	(*Part 37 Present*)
		Part_Present37FB(
			Sensor_Input:= N08.I.4,
			On_Trigger1:= Enable_Motion AND In_Auto AND NOT Unload_Complete,
			On_Trigger2:= TRUE,
			Off_Trigger1:= Dry_Cycle OR (Cycle_Complete  AND NOT Enable_Motion),
			Off_Trigger2:= TRUE,
			Disable_Faults:= FALSE,
			Fault_Delay:= T#1.5s,
			Status=> Part_Present37,
			Faulted=>  PPFaults1.8);

	(*Part 38 Present*)
		Part_Present38FB(
			Sensor_Input:= N08.I.5,
			On_Trigger1:= Enable_Motion AND In_Auto AND NOT Unload_Complete,
			On_Trigger2:= TRUE,
			Off_Trigger1:= Dry_Cycle OR (Cycle_Complete  AND NOT Enable_Motion),
			Off_Trigger2:= TRUE,
			Disable_Faults:= FALSE,
			Fault_Delay:= T#1.5s,
			Status=> Part_Present38,
			Faulted=>  PPFaults1.9);

	(*Part 39 Present*)
		Part_Present39FB(
			Sensor_Input:= N08.I.6,
			On_Trigger1:= Enable_Motion AND In_Auto AND NOT Unload_Complete,
			On_Trigger2:= TRUE,
			Off_Trigger1:= Dry_Cycle OR (Cycle_Complete  AND NOT Enable_Motion),
			Off_Trigger2:= TRUE,
			Disable_Faults:= FALSE,
			Fault_Delay:= T#1.5s,
			Status=> Part_Present39,
			Faulted=>  PPFaults1.10);

	(*Part 40 Present*)
		Part_Present40FB(
			Sensor_Input:= N08.I.7,
			On_Trigger1:= Enable_Motion AND In_Auto AND NOT Unload_Complete,
			On_Trigger2:= TRUE,
			Off_Trigger1:= Dry_Cycle OR (Cycle_Complete  AND NOT Enable_Motion),
			Off_Trigger2:= TRUE,
			Disable_Faults:= FALSE,
			Fault_Delay:= T#1.5s,
			Status=> Part_Present40,
			Faulted=>  PPFaults1.11);



(*end*)
END_ACTION

ACTION Robot_Registration:


(*#################################### Register Robots to Tool ##################################*)
(*+++++++++++THIS AREA IS CUSTOM PER INSTALLATION AND WILL HAVE TO BE MODIFIED PER +++++++++++++*)
(*+++++++++++THIS AREA IS CUSTOM PER INSTALLATION AND WILL HAVE TO BE MODIFIED PER +++++++++++++*)
(*NOTE: See Example code in Fix 15 / 16*)
(*NOTE: See Example code in Fix 15 / 16*)

	(*Data From Load Robot(s)*)
	Load_Robots_Clear1:= TRUE;
	Load_Robots_Clear2:= TRUE;
	Load_Robots_Clear:=Load_Robots_Clear1 AND Load_Robots_Clear2;
	Load_Robots_WorkingOK1:= FALSE;
	Load_Robots_WorkingOK2:= FALSE;
	IF FALSE
		THEN
		Load_Robots_UnclampEarly1:= TRUE;
	END_IF;
	IF FALSE
		THEN
		Load_Robots_UnclampEarly2:= TRUE;
	END_IF;
	Load_Robots_Complete1:= FALSE;
	Load_Robots_Complete2:= FALSE;
	Load_Robots_PartInEOAT1:= FALSE;
	Load_Robots_PartInEOAT2:= FALSE;


	(*Data From Turntable*)
	TurntableA_Clear:= TRUE;
	TurntableB_Clear:= TRUE;
	Turntable_Clear:= TurntableA_Clear AND TurntableB_Clear;
	TurntableA_At_Robot:= FALSE;
	TurntableB_At_Robot:= FALSE;
	Turntable_WorkingOK:= FALSE;
	TurntableA_Complete:= FALSE;
	TurntableB_Complete:= FALSE;


	(*Data From Seal Robot(s)*)
	Seal_Robots_Clear:= TRUE;
	Seal_Robots_WorkingOK:= FALSE;
	IF FALSE
		THEN
		Seal_Robots_UnclampEarly:= TRUE;
	END_IF;
	Seal_Robots_Complete:= FALSE;


	(*Data From Stud Robot(s)*)
	Stud_Robots_Clear:= TRUE;
	Stud_Robots_WorkingOK:= FALSE;
	IF FALSE
		THEN
		Stud_Robots_UnclampEarly:= TRUE;
	END_IF;
	Stud_Robots_Complete:= FALSE;


	(*Data From Weld Robot(s)*)
	Weld_Robots_Clear:= TRUE;
	Weld_Robots_WorkingOK:= FALSE;
	IF FALSE
		THEN
		Weld_Robots_UnclampEarly:= TRUE;
	END_IF;
	Weld_Robots_Complete:= FALSE;

	(*Change Robots for Current Fixture functionality*) (*If no MIG robots Set to True.  Example code is in Fix15/16*) 
	Mig_Robots_Ready:=	TRUE; 

	(*Data From Unload Robot(s)*)
	Unload_Robots_Clear1:= TRUE;
	Unload_Robots_Clear2:= TRUE;
	Unload_Robots_Clear:= Unload_Robots_Clear1 AND Unload_Robots_Clear2;
	Unload_Robots_WorkingOK1:= FALSE;
	Unload_Robots_WorkingOK2:= FALSE;
	Unload_Robots_Complete1:= FALSE;
	Unload_Robots_Complete2:= FALSE;
	Unload_Robots_EOATEmpty1:=FALSE;
	Unload_Robots_EOATEmpty2:= FALSE;



	(*Amalgumate All Robots Clear of Tool*)
	All_Robots_Clear:= Load_Robots_Clear AND Seal_Robots_Clear AND Stud_Robots_Clear AND Turntable_Clear AND Weld_Robots_Clear AND Unload_Robots_Clear;

	(*Data To All Robots*)
	(*Task ID*)
	R1_Data.Task_ID[1]:=Task_ID;

	(*Fix ID*)
	R1_Data.Fix_ID[1]:=Fix_ID;

	(*Model ID*)
	R1_Data.Model_ID[1]:=Model_ID;

	(*Proceed from Pounce*)
	R1_Data.Proceed_From_Pounce[1]:= Robots_Clear_ToProceed;

	(*Complete Acks*)
	R1_Data.Complete_Ack[1]:=(Weld_Complete_Ack AND Weld_Robots_WorkingOK);

	(*Repo Acks*)
	R1_Data.PeripheralReq_Ack[1]:= Repo_Ack;

(*%%%%%%%%%%%%%% Call Robots to Tool and Give Them, Task ID, Fixture ID and Model ID %%%%%%%%%%%%%%%%%*)
	(* Perform Call To Tool*)
	Tool_Call_ForLoadRobots1:= Enable_Motion AND (NOT Cell_In_Services OR NOT Load_Robots_Clear1)
						AND Start_Load_Robots1 AND NOT Start_Load_Robots2 AND NOT Start_Weld_Robots AND NOT Start_Seal_Robots AND NOT Start_Stud_Robots
						AND NOT Start_Unload_Robots1 AND NOT Start_Unload_Robots2 AND NOT Start_TurntableA AND NOT Start_TurntableB;
	Tool_Call_ForLoadRobots2:= Enable_Motion AND (NOT Cell_In_Services OR NOT Load_Robots_Clear2)
						AND NOT Start_Load_Robots1 AND Start_Load_Robots2 AND NOT Start_Weld_Robots AND NOT Start_Seal_Robots AND NOT Start_Stud_Robots
						AND NOT Start_Unload_Robots1 AND NOT Start_Unload_Robots2 AND NOT Start_TurntableA AND NOT Start_TurntableB;
	Tool_Call_ForSealRobots:=Enable_Motion AND (NOT Cell_In_Services OR NOT Seal_Robots_Clear)
						AND NOT Start_Load_Robots1 AND NOT Start_Load_Robots2 AND NOT Start_Weld_Robots AND Start_Seal_Robots AND NOT Start_Stud_Robots
						AND NOT Start_Unload_Robots1 AND NOT Start_Unload_Robots2 AND NOT Start_TurntableA AND NOT Start_TurntableB;
	Tool_Call_ForStudRobots:=Enable_Motion AND (NOT Cell_In_Services OR NOT Stud_Robots_Clear)
						AND NOT Start_Load_Robots1 AND NOT Start_Load_Robots2 AND NOT Start_Weld_Robots AND NOT Start_Seal_Robots AND Start_Stud_Robots
						AND NOT Start_Unload_Robots1 AND NOT Start_Unload_Robots2 AND NOT Start_TurntableA AND NOT Start_TurntableB;
	Tool_Call_ForSweepA:= Enable_Motion AND (NOT Cell_In_Services OR NOT TurntableA_Clear)
						AND NOT Start_Load_Robots1 AND NOT Start_Load_Robots2 AND NOT Start_Weld_Robots AND NOT Start_Seal_Robots AND NOT Start_Stud_Robots
						AND NOT Start_Unload_Robots1 AND NOT Start_Unload_Robots2 AND Start_TurntableA AND NOT Start_TurntableB;
	Tool_Call_ForSweepB:= Enable_Motion AND (NOT Cell_In_Services OR NOT TurntableB_Clear)
						AND NOT Start_Load_Robots1 AND NOT Start_Load_Robots2 AND NOT Start_Weld_Robots AND NOT Start_Seal_Robots AND NOT Start_Stud_Robots
						AND NOT Start_Unload_Robots1 AND NOT Start_Unload_Robots2 AND NOT Start_TurntableA AND Start_TurntableB;
	Tool_Call_ForWeldRobots:= Enable_Motion AND (NOT Cell_In_Services OR NOT Weld_Robots_Clear)
						AND NOT Start_Load_Robots1 AND NOT Start_Load_Robots2 AND Start_Weld_Robots AND NOT Start_Seal_Robots AND NOT Start_Stud_Robots
						AND NOT Start_Unload_Robots1 AND NOT Start_Unload_Robots2 AND NOT Start_TurntableA AND NOT Start_TurntableB;
	Tool_Call_ForUnloadRobots1:= Enable_Motion AND (NOT Cell_In_Services OR NOT Unload_Robots_Clear1)
						AND NOT Start_Load_Robots1 AND NOT Start_Load_Robots2 AND NOT Start_Weld_Robots AND NOT Start_Seal_Robots AND NOT Start_Stud_Robots
						AND Start_Unload_Robots1 AND NOT Start_Unload_Robots2 AND NOT Start_TurntableA AND NOT Start_TurntableB;
	Tool_Call_ForUnloadRobots2:= Enable_Motion AND (NOT Cell_In_Services OR NOT Unload_Robots_Clear2)
						AND NOT Start_Load_Robots1 AND NOT Start_Load_Robots2 AND NOT Start_Weld_Robots AND NOT Start_Seal_Robots AND NOT Start_Stud_Robots
						AND NOT Start_Unload_Robots1 AND Start_Unload_Robots2 AND NOT Start_TurntableA AND NOT Start_TurntableB;



	(*Allow Robots to Proceed Into Tool*)
	(*!!!!!This is the final OK to allow Robots Into the Tool Area, So it Better Be Ready!!!!!!!*)
	IF Enable_Motion
		THEN
			IF Load_Robots_Proceed1 AND Load_Robots_WorkingOK1 AND Load_Robots_Clear2 AND Seal_Robots_Clear AND Stud_Robots_Clear AND Turntable_Clear AND Weld_Robots_Clear AND Unload_Robots_Clear
				THEN Robots_Clear_ToProceed:=TRUE;
			ELSIF Load_Robots_Proceed2 AND Load_Robots_WorkingOK2 AND Load_Robots_Clear1 AND Seal_Robots_Clear AND Stud_Robots_Clear AND Turntable_Clear AND Weld_Robots_Clear AND Unload_Robots_Clear
				THEN Robots_Clear_ToProceed:=TRUE;
			ELSIF Seal_Robots_Proceed AND Seal_Robots_WorkingOK AND Load_Robots_Clear AND Stud_Robots_Clear AND Turntable_Clear AND Weld_Robots_Clear AND Unload_Robots_Clear
				THEN Robots_Clear_ToProceed:=TRUE;
			ELSIF Stud_Robots_Proceed AND Stud_Robots_WorkingOK AND Load_Robots_Clear AND Seal_Robots_Clear AND Turntable_Clear AND Weld_Robots_Clear AND Unload_Robots_Clear
				THEN Robots_Clear_ToProceed:=TRUE;
			ELSIF Weld_Robots_Proceed AND Weld_Robots_WorkingOK AND Load_Robots_Clear AND Seal_Robots_Clear AND Stud_Robots_Clear AND Turntable_Clear AND Unload_Robots_Clear
				THEN Robots_Clear_ToProceed:=TRUE;
			ELSIF Unload_Robots_Proceed1 AND Unload_Robots_WorkingOK1 AND Load_Robots_Clear AND Seal_Robots_Clear AND Stud_Robots_Clear AND Turntable_Clear AND Weld_Robots_Clear AND Unload_Robots_Clear2
				THEN Robots_Clear_ToProceed:=TRUE;
			ELSIF Unload_Robots_Proceed2 AND Unload_Robots_WorkingOK2 AND Load_Robots_Clear AND Seal_Robots_Clear AND Stud_Robots_Clear AND Turntable_Clear AND Weld_Robots_Clear AND Unload_Robots_Clear1
				THEN Robots_Clear_ToProceed:=TRUE;
			ELSE Robots_Clear_ToProceed:= FALSE;
			END_IF;
		ELSE Robots_Clear_ToProceed:= FALSE;
	END_IF;

(*+++++++++++++++++++++++++++++++++++++++++++++++ Task Complete Acks ++++++++++++++++++++++++++*)
	(*1st Load Complete Ack*)
	Load_Complete1_Ack:= Load_Robots_Complete1 AND Load_Complete1;

	(*2nd Load Complete Ack*)
	Load_Complete2_Ack:= Load_Robots_Complete2 AND Load_Complete2;

	(*Seal Complete Ack*)
	Seal_Complete_Ack:= Seal_Robots_Complete AND Sealing_Complete;

	(*Stud Complete Ack*)
	Stud_Complete_Ack:= Stud_Robots_Complete AND Stud_Complete;

	(*Sweep Complete ACK*)
	TurnA_Complete_Ack := TurntableA_Complete AND TurntableA_At_Robot;
	TurnB_Complete_Ack := TurntableB_Complete AND TurntableB_At_Robot;

	(*Weld Complete Ack*)
	Weld_Complete_Ack:= Weld_Robots_Complete AND Welding_Complete;

	(*Unload Complete Ack*)
	Unload_Complete1_Ack:= Unload_Robots_Complete1 AND Unload_Complete;

	(*Unload Complete Ack*)
	Unload_Complete2_Ack:= Unload_Robots_Complete2 AND Unload_Complete;







(*end*)
END_ACTION

ACTION Status_and_Faults:



(*^^^^^^^^^^^^^^^^^^^^^^^^^^^^^^^^^^^^^^ General Visualization ^^^^^^^^^^^^^^^^^^^^^^^^^^^^^^^^^^^^*)
	(*For Ready to Load Indicators*)
		(*Flash when tool should be loaded but load is not complete*)
		IF In_Auto AND Tool_At_Home AND NOT Welding_Complete AND All_Robots_Clear AND NOT All_Sensors_On.2
			THEN
				Ready_To_Load:= Pulse_500mS;
				(*Go solid when tool has been loaded properly*)
				(*Go solid when tool is ready to be unloaded*)
		ELSIF In_Auto AND All_Robots_Clear  AND ((Tool_At_Home AND NOT Welding_Complete AND All_Sensors_On.2 AND NOT Enable_Motion)
			OR (Tool_At_Unload.0 AND Welding_Complete AND (Sealing_Complete OR Sealer_Bypass) AND (Stud_Complete OR Stud_Bypass) AND TurntableA_At_Robot AND NOT All_Sensors_Off))
			THEN
				Ready_To_Load:= TRUE;
		ELSE
				Ready_To_Load:= FALSE;
		END_IF;
	(*For Red Stack Light Indicators*)
		Red_Lamp_Req:= PPFaults<>0 OR CLFaulted.0 OR CLFaulted.4 OR (NOT Sealer_Bypass AND MAIN.SL01.Disp1_Volume_NotOK AND (MAIN.R1.Task_ID_Ack=Seal_Fix01)) OR Load_Seq01.Faulted;


	(*Status Banners*)
		(*1 - Check Parts On Sub Check*)
		IF In_Auto AND NOT In_Manual AND NOT Cycle_Complete AND Tool_At_Load.0
			AND NOT Start_Load_Robots1 AND NOT Start_Load_Robots2 AND NOT Start_Seal_Robots AND NOT Start_Stud_Robots AND NOT Start_TurntableA
			AND NOT Start_TurntableB AND NOT Start_Weld_Robots AND NOT Start_Unload_Robots1 AND NOT Start_Unload_Robots2
			THEN
				IF NOT Dry_Cycle AND NOT All_Sensors_On.0
					THEN Status:= 1;
				ELSIF Dry_Cycle AND NOT Load_Complete1
					THEN Status:=1;
				END_IF;
		END_IF;
		(*2 - Sub Check OK*)
		IF In_Auto AND NOT In_Manual AND NOT Cycle_Complete AND Tool_At_Load.1
			AND NOT Start_Load_Robots1 AND NOT Start_Load_Robots2 AND NOT Start_Seal_Robots AND NOT Start_Stud_Robots AND NOT Start_TurntableA
			AND NOT Start_TurntableB AND NOT Start_Weld_Robots AND NOT Start_Unload_Robots1 AND NOT Start_Unload_Robots2
			THEN
				IF NOT Dry_Cycle AND NOT All_Sensors_On.1
					THEN Status:= 2;
				ELSIF Dry_Cycle AND NOT Load_Complete2
					THEN Status:=2;
				END_IF;
		END_IF;
		(*3 - Load Main Part*)
		IF In_Auto AND NOT In_Manual AND NOT Cycle_Complete AND Tool_At_Home
			AND NOT Start_Load_Robots1 AND NOT Start_Load_Robots2 AND NOT Start_Seal_Robots AND NOT Start_Stud_Robots AND NOT Start_TurntableA
			AND NOT Start_TurntableB AND NOT Start_Weld_Robots AND NOT Start_Unload_Robots1 AND NOT Start_Unload_Robots2
			THEN
				IF NOT Dry_Cycle AND NOT All_Sensors_On.2
					THEN Status:= 3;
				ELSIF Dry_Cycle AND NOT Load_Complete
					THEN Status:=3;
				END_IF;
		END_IF;
		(*10 - Load Parts Onto Tool*)
		IF In_Auto AND NOT In_Manual AND NOT Cycle_Complete AND Tool_At_Load.0
			AND NOT Start_Load_Robots1 AND NOT Start_Load_Robots2 AND NOT Start_Seal_Robots AND NOT Start_Stud_Robots AND NOT Start_TurntableA
			AND NOT Start_TurntableB AND NOT Start_Weld_Robots AND NOT Start_Unload_Robots1 AND NOT Start_Unload_Robots2
			THEN
				IF NOT Dry_Cycle AND NOT All_Sensors_On.2
					THEN Status:= 10;
				ELSIF Dry_Cycle AND NOT Load_Complete
					THEN Status:=10;
				END_IF;
		END_IF;
		(*11 - Robot(s) Loading*)
		IF ((Start_Load_Robots1 OR  Load_Robots_WorkingOK1) OR (Start_Load_Robots2 OR  Load_Robots_WorkingOK2)) AND In_Auto AND NOT In_Manual
			AND NOT Start_Seal_Robots AND NOT Start_Stud_Robots AND NOT Start_TurntableA
			AND NOT Start_TurntableB AND NOT Start_Weld_Robots AND NOT Start_Unload_Robots1 AND NOT Start_Unload_Robots2
			THEN Status:= 11;
		END_IF;
		(*12 - Parts Loaded OK*)
		IF In_Auto AND NOT In_Manual AND NOT Cycle_Complete
			AND NOT Start_Load_Robots1 AND NOT Start_Load_Robots2 AND NOT Start_Seal_Robots AND NOT Start_Stud_Robots AND NOT Start_TurntableA
			 AND NOT Start_TurntableB AND NOT Start_Weld_Robots AND NOT Start_Unload_Robots1 AND NOT Start_Unload_Robots2
			THEN
				IF (All_Sensors_On.2 AND Tool_At_Load.0) AND NOT Dry_Cycle
					THEN Status:= 12;
				ELSIF Load_Complete
					THEN Status:= 12;
				END_IF;
		END_IF;
		(*19 - Robot(s) Stud*)
		IF (Start_Stud_Robots OR Stud_Robots_WorkingOK) AND In_Auto AND NOT In_Manual
			AND NOT Start_Load_Robots1 AND NOT Start_Load_Robots2 AND NOT Start_Weld_Robots AND NOT Start_Seal_Robots AND NOT Start_TurntableA
			 AND NOT Start_TurntableB AND NOT Start_Unload_Robots1 AND NOT Start_Unload_Robots2
			THEN Status:= 19;
		END_IF;
		(*20 - Robot(s) Sealing*)
		IF (Start_Seal_Robots OR Seal_Robots_WorkingOK) AND In_Auto AND NOT In_Manual
			AND NOT Start_Load_Robots1 AND NOT Start_Load_Robots2 AND NOT Start_Weld_Robots AND NOT Start_Stud_Robots AND NOT Start_TurntableA
			 AND NOT Start_TurntableB AND NOT Start_Unload_Robots1 AND NOT Start_Unload_Robots2
			THEN Status:= 20;
		END_IF;
		(*21 - Robot(s) Welding*)
		IF (Start_Weld_Robots OR Weld_Robots_WorkingOK) AND In_Auto AND NOT In_Manual
			AND NOT Start_Load_Robots1 AND NOT Start_Load_Robots2 AND NOT Start_Seal_Robots AND NOT Start_Stud_Robots AND NOT Start_TurntableA
			 AND NOT Start_TurntableB AND NOT Start_Unload_Robots1 AND NOT Start_Unload_Robots2
			THEN Status:= 21;
		END_IF;
		(*22 - Welding Complete / Ready for Unload*)
		IF In_Auto AND NOT In_Manual AND NOT Cycle_Complete AND Welding_Complete
			AND NOT Start_Load_Robots1 AND NOT Start_Load_Robots2 AND NOT Start_Seal_Robots AND NOT Start_Stud_Robots AND NOT Start_TurntableA
			AND NOT Start_TurntableB AND NOT Start_Weld_Robots AND NOT Start_Unload_Robots1 AND NOT Start_Unload_Robots2
			THEN Status:= 22;
		END_IF;
		(*26 - Ready for Rotate*)
		IF (Start_TurntableA OR Start_TurntableB) AND In_Auto AND NOT In_Manual
			AND NOT Start_Load_Robots1 AND NOT Start_Load_Robots2 AND NOT Start_Seal_Robots AND NOT Start_Stud_Robots
			AND NOT Start_Weld_Robots AND NOT Start_Unload_Robots1 AND NOT Start_Unload_Robots2
			THEN Status := 26;
		END_IF;
		(*31 - Robot(s) Unloading*)
		IF (Start_Unload_Robots1 OR Unload_Robots_WorkingOK1 OR Start_Unload_Robots2 OR Unload_Robots_WorkingOK2) AND In_Auto AND NOT In_Manual
			AND NOT Start_Load_Robots1 AND NOT Start_Load_Robots2 AND NOT Start_Seal_Robots AND NOT Start_Stud_Robots AND NOT Start_TurntableA
			AND NOT Start_TurntableB AND NOT Start_Weld_Robots
			THEN Status:= 31;
		END_IF;
		(*32 - Unload Complete*)
		IF In_Auto AND NOT In_Manual AND NOT Cycle_Complete AND Unload_Complete
			AND NOT Start_Load_Robots1 AND NOT Start_Load_Robots2 AND NOT Start_Seal_Robots AND NOT Start_Stud_Robots AND NOT Start_TurntableA
			AND NOT Start_TurntableB AND NOT Start_Weld_Robots AND NOT Start_Unload_Robots1 AND NOT Start_Unload_Robots2
			THEN Status:= 32;
		END_IF;
		(*42 - Cycle Complete*)
		IF In_Auto AND NOT In_Manual AND Cycle_Complete AND All_Sensors_Off
			THEN Status:= 42;
		END_IF;
		(*50 - In Manual*)
		IF In_Manual
			THEN Status:= 50;
		END_IF;
		(*51 - Clamp Fault*)
		IF (CLFaults1>0 OR CLFaults2>0 OR CLFaults3>0 OR CLFaults4>0) AND In_Auto AND NOT In_Manual
			THEN Status:= 51;
		END_IF;
		(*52 - Part Present Sensor Fault*)
		IF PPFaults>0 AND In_Auto AND NOT In_Manual
			THEN Status:= 52;
		END_IF;
		(*53 - Nut Checks Failed Call QA*)
		IF QAChecks_Failed AND In_Auto AND NOT In_Manual
			THEN Status:= 53;
		END_IF;
		(*54 - Sealer Failed Call QA*)
		IF NOT Sealer_Bypass AND (MAIN.SL01.Disp1_Volume_NotOK AND (MAIN.R1.Task_ID_Ack=Seal_Fix01)) AND In_Auto AND NOT In_Manual
			THEN Status:= 54;
		END_IF;
		(*55 - Load Sequence Fault Call QA*)
		IF Load_Seq01.Faulted AND In_Auto AND NOT In_Manual
			THEN Status:= 55;
		END_IF;



(*$$$$$$$$$$$$$$$$$$$$$$$$$$$$$$$$$$$$$$$$$$$$$$$$$$$ Faults $$$$$$$$$$$$$$$$$$$$$$$$$$$$$$$$$$$$$$$$$$$$$$$$$$$$$$$*)

	(*Clamp/Cylider Faults Group 1*)
		IF CLFaults1>0
			THEN CLFaulted.1:=TRUE;
		ELSE
			CLFaulted.1:=FALSE;
		END_IF;
	(*Clamp/Cylider Faults Group 2*)
		IF CLFaults2>0
			THEN CLFaulted.2:=TRUE;
		ELSE
			CLFaulted.2:=FALSE;
		END_IF;
	(*Clamp/Cylider Faults Group 3*)
		IF CLFaults3>0
			THEN CLFaulted.3:=TRUE;
		ELSE
			CLFaulted.3:=FALSE;
		END_IF;
	(*Clamp/Cylinder Faults Group 4 - Reserved Flag for QA Check Motion Faults*)
		IF CLFaults4>0
			THEN CLFaulted.4:=TRUE;
		ELSE
			CLFaulted.4:=FALSE;
		END_IF;
	(*Bit 0 is designated as ANY Clamp Group Faulted*)
	IF CLFaulted.1 OR CLFaulted.2 OR CLFaulted.3
		THEN CLFaulted.0:= TRUE;
	ELSE CLFaulted.0 := FALSE;
	END_IF;

	(*Part Present Sensor Faults*)
		IF (PPFaults>0) OR (PPFaults1>0) OR (PPFaults2>0)
			THEN PPFaulted.0:=TRUE;
		ELSE
			PPFaulted.0:=FALSE;
		END_IF;
























(*end*)
END_ACTION

ACTION Task_Fix_Model_IDs:


	(*Develop Task IDs - See Global Variable, "TaskID_Record"*)

	IF (Start_Load_Robots1 OR Start_Load_Robots2) AND Enable_Motion
		THEN Task_ID:= Dropoff_Fix12;
	ELSIF Start_Seal_Robots AND Enable_Motion
		THEN Task_ID:= Seal_Fix12;
	ELSIF Start_Stud_Robots AND Enable_Motion
		THEN Task_ID:= Stud_Fix12;
	ELSIF Start_Weld_Robots AND Enable_Motion
		THEN Task_ID:= Weld_Fix12;
	ELSIF Start_TurnTableA AND Enable_Motion
		THEN Task_ID:= Sweep_Fix12;
	ELSIF (Start_Unload_Robots1 OR Start_Unload_Robots2) AND Enable_Motion
		THEN Task_ID:= Pickup_Fix12;
	ELSE Task_ID:= 0;
	END_IF;

	(*Develop Fixture ID*)
	Fix_ID:= N00.ID;					(*In Future Map Beckhoff Dip Switch Data From IP67 Block to Here*)

	(*Develop Model ID*)
	Model_ID:= Discrete_In.ModelData;
END_ACTION

ACTION Tool_States:


(*+++++++++++THIS AREA IS CUSTOM PER INSTALLATION AND WILL HAVE TO BE MODIFIED PER +++++++++++++*)
(*+++++++++++THIS AREA IS CUSTOM PER INSTALLATION AND WILL HAVE TO BE MODIFIED PER +++++++++++++*)

	Tool_At_HOME:= Clamp1RETD AND Clamp2RETD AND Clamp3RETD AND Clamp4RETD
				AND Clamp5RETD AND Clamp6RETD AND Clamp7RETD AND Clamp8RETD
				AND Clamp9RETD AND Clamp10RETD AND Clamp11RETD AND Clamp12RETD
				AND Clamp13RETD AND Clamp14RETD AND Clamp15RETD AND Clamp16RETD
				AND Clamp17RETD AND Clamp18RETD AND Clamp19RETD AND Clamp20RETD
				AND Clamp21RETD AND Clamp22RETD AND Clamp23RETD AND Clamp24RETD
				AND Pin1ADVD AND Pin2ADVD AND Pin3ADVD AND Pin4ADVD AND Pin5ADVD AND Pin6ADVD AND Pin7ADVD
				AND Pin8ADVD AND Pin9ADVD AND Pin10ADVD AND Pin11ADVD AND Pin12ADVD AND Pin13ADVD AND Pin14ADVD
				AND Slide1RETD AND Slide2RETD AND Slide3RETD AND Slide4RETD AND Slide5RETD AND Slide6RETD
				AND Swing1ADVD AND Swing2ADVD AND Swing3ADVD AND Swing4ADVD AND Swing5ADVD AND Swing6ADVD;


	Tool_At_Load.0:=Clamp1RETD AND Clamp2RETD AND Clamp3RETD AND Clamp4RETD
				AND Clamp5RETD AND Clamp6RETD AND Clamp7RETD AND Clamp8RETD
				AND Clamp9RETD AND Clamp10RETD AND Clamp11RETD AND Clamp12RETD
				AND Clamp13RETD AND Clamp14RETD AND Clamp15RETD AND Clamp16RETD
				AND Clamp17RETD AND Clamp18RETD AND Clamp19RETD AND Clamp20RETD
				AND Clamp21RETD AND Clamp22RETD AND Clamp23RETD AND Clamp24RETD
				AND Pin1ADVD AND Pin2ADVD AND Pin3ADVD AND Pin4ADVD AND Pin5ADVD AND Pin6ADVD AND Pin7ADVD
				AND Pin8ADVD AND Pin9ADVD AND Pin10ADVD AND Pin11ADVD AND Pin12ADVD AND Pin13ADVD AND Pin14ADVD
				AND Slide1RETD AND Slide2RETD AND Slide3RETD AND Slide4RETD AND Slide5RETD AND Slide6RETD
				AND Swing1ADVD AND Swing2ADVD AND Swing3ADVD AND Swing4ADVD AND Swing5ADVD AND Swing6ADVD;
	Tool_At_Load.1:=FALSE;
	Tool_At_Load.2:= FALSE;
	Tool_At_Load.3:= FALSE;
	Tool_At_Load.4:= FALSE;


	Tool_At_Seal.0:= Clamp1ADVD AND Clamp2ADVD AND Clamp3ADVD AND Clamp4ADVD
				AND Clamp5ADVD AND Clamp6ADVD AND Clamp7ADVD AND Clamp8ADVD
				AND Clamp9ADVD AND Clamp10ADVD AND Clamp11ADVD AND Clamp12ADVD
				AND Clamp13ADVD AND Clamp14ADVD AND Clamp15ADVD AND Clamp16ADVD
				AND Clamp17ADVD AND Clamp18ADVD AND Clamp19ADVD AND Clamp20ADVD
				AND Clamp21ADVD AND Clamp22ADVD AND Clamp23ADVD AND Clamp24ADVD
				AND Pin1ADVD AND Pin2ADVD AND Pin3ADVD AND Pin4ADVD AND Pin5ADVD AND Pin6ADVD AND Pin7ADVD
				AND Pin8ADVD AND Pin9ADVD AND Pin10ADVD AND Pin11ADVD AND Pin12ADVD AND Pin13ADVD AND Pin14ADVD
				AND Slide1RETD AND Slide2RETD AND Slide3RETD AND Slide4RETD AND Slide5RETD AND Slide6RETD
				AND Swing1ADVD AND Swing2ADVD AND Swing3ADVD AND Swing4ADVD AND Swing5ADVD AND Swing6ADVD;
	Tool_At_Seal.1:= FALSE;
	Tool_At_Seal.2:= FALSE;
	Tool_At_Seal.3:= FALSE;
	Tool_At_Seal.4:= FALSE;


	Tool_At_Stud.0:= Clamp1ADVD AND Clamp2ADVD AND Clamp3ADVD AND Clamp4ADVD
				AND Clamp5ADVD AND Clamp6ADVD AND Clamp7ADVD AND Clamp8ADVD
				AND Clamp9ADVD AND Clamp10ADVD AND Clamp11ADVD AND Clamp12ADVD
				AND Clamp13ADVD AND Clamp14ADVD AND Clamp15ADVD AND Clamp16ADVD
				AND Clamp17ADVD AND Clamp18ADVD AND Clamp19ADVD AND Clamp20ADVD
				AND Clamp21ADVD AND Clamp22ADVD AND Clamp23ADVD AND Clamp24ADVD
				AND Pin1ADVD AND Pin2ADVD AND Pin3ADVD AND Pin4ADVD AND Pin5ADVD AND Pin6ADVD AND Pin7ADVD
				AND Pin8ADVD AND Pin9ADVD AND Pin10ADVD AND Pin11ADVD AND Pin12ADVD AND Pin13ADVD AND Pin14ADVD
				AND Slide1RETD AND Slide2RETD AND Slide3RETD AND Slide4RETD AND Slide5RETD AND Slide6RETD
				AND Swing1ADVD AND Swing2ADVD AND Swing3ADVD AND Swing4ADVD AND Swing5ADVD AND Swing6ADVD;
	Tool_At_Stud.1:= FALSE;
	Tool_At_Stud.2:= FALSE;
	Tool_At_Stud.3:= FALSE;
	Tool_At_Stud.4:= FALSE;


	Tool_At_Rotate.0:= Clamp1ADVD AND Clamp2ADVD AND Clamp3ADVD AND Clamp4ADVD
				AND Clamp5ADVD AND Clamp6ADVD AND Clamp7ADVD AND Clamp8ADVD
				AND Clamp9ADVD AND Clamp10ADVD AND Clamp11ADVD AND Clamp12ADVD
				AND Clamp13ADVD AND Clamp14ADVD AND Clamp15ADVD AND Clamp16ADVD
				AND Clamp17ADVD AND Clamp18ADVD AND Clamp19ADVD AND Clamp20ADVD
				AND Clamp21ADVD AND Clamp22ADVD AND Clamp23ADVD AND Clamp24ADVD
				AND Pin1ADVD AND Pin2ADVD AND Pin3ADVD AND Pin4ADVD AND Pin5ADVD AND Pin6ADVD AND Pin7ADVD
				AND Pin8ADVD AND Pin9ADVD AND Pin10ADVD AND Pin11ADVD AND Pin12ADVD AND Pin13ADVD AND Pin14ADVD
				AND Slide1RETD AND Slide2RETD AND Slide3RETD AND Slide4RETD AND Slide5RETD AND Slide6RETD
				AND Swing1ADVD AND Swing2ADVD AND Swing3ADVD AND Swing4ADVD AND Swing5ADVD AND Swing6ADVD;
	Tool_At_Rotate.1:= FALSE;
	Tool_At_Rotate.2:= FALSE;
	Tool_At_Rotate.3:= FALSE;
	Tool_At_Rotate.4:= FALSE;


	Tool_At_Weld.0:= Clamp1ADVD AND Clamp2ADVD AND Clamp3ADVD AND Clamp4ADVD
				AND Clamp5ADVD AND Clamp6ADVD AND Clamp7ADVD AND Clamp8ADVD
				AND Clamp9ADVD AND Clamp10ADVD AND Clamp11ADVD AND Clamp12ADVD
				AND Clamp13ADVD AND Clamp14ADVD AND Clamp15ADVD AND Clamp16ADVD
				AND Clamp17ADVD AND Clamp18ADVD AND Clamp19ADVD AND Clamp20ADVD
				AND Clamp21ADVD AND Clamp22ADVD AND Clamp23ADVD AND Clamp24ADVD
				AND Pin1ADVD AND Pin2ADVD AND Pin3ADVD AND Pin4ADVD AND Pin5ADVD AND Pin6ADVD AND Pin7ADVD
				AND Pin8ADVD AND Pin9ADVD AND Pin10ADVD AND Pin11ADVD AND Pin12ADVD AND Pin13ADVD AND Pin14ADVD
				AND Slide1RETD AND Slide2RETD AND Slide3RETD AND Slide4RETD AND Slide5RETD AND Slide6RETD
				AND Swing1ADVD AND Swing2ADVD AND Swing3ADVD AND Swing4ADVD AND Swing5ADVD AND Swing6ADVD;
	Tool_At_Weld.1:= FALSE;
	Tool_At_Weld.2:= FALSE;
	Tool_At_Weld.3:= FALSE;
	Tool_At_Weld.4:= FALSE;


	Tool_At_Unload.0:=Clamp1RETD AND Clamp2RETD AND Clamp3RETD AND Clamp4RETD
				AND Clamp5RETD AND Clamp6RETD AND Clamp7RETD AND Clamp8RETD
				AND Clamp9RETD AND Clamp10RETD AND Clamp11RETD AND Clamp12RETD
				AND Clamp13RETD AND Clamp14RETD AND Clamp15RETD AND Clamp16RETD
				AND Clamp17RETD AND Clamp18RETD AND Clamp19RETD AND Clamp20RETD
				AND Clamp21RETD AND Clamp22RETD AND Clamp23RETD AND Clamp24RETD
				AND Pin1RETD AND Pin2RETD AND Pin3RETD AND Pin4RETD AND Pin5RETD AND Pin6RETD AND Pin7RETD
				AND Pin8RETD AND Pin9RETD AND Pin10RETD AND Pin11RETD AND Pin12RETD AND Pin13RETD AND Pin14RETD
				AND Slide1ADVD AND Slide2ADVD AND Slide3ADVD AND Slide4ADVD AND Slide5ADVD AND Slide6ADVD
				AND Swing1RETD AND Swing2RETD AND Swing3RETD AND Swing4RETD AND Swing5RETD AND Swing6RETD;
	Tool_At_Unload.1:=FALSE;
	Tool_At_Unload.2:= FALSE;
	Tool_At_Unload.3:= FALSE;
	Tool_At_Unload.4:= FALSE;







































(*end*)
END_ACTION

ACTION Tool_VBSeq_Repos:
(*+++++++++++THIS AREA IS CUSTOM PER INSTALLATION AND WILL HAVE TO BE MODIFIED PER +++++++++++++*)
(*+++++++++++THIS AREA IS CUSTOM PER INSTALLATION AND WILL HAVE TO BE MODIFIED PER +++++++++++++*)


(*!!!!!!!!!!!!!!!!!!!!!!!!!!!!!!!!!!!!!!!!!! Tool Motion Control !!!!!!!!!!!!!!!!!!!!!!!!!!!!!!!*)

(*----------------------------------------- Camp / Unclamp Steps -------------------------------*)

(*$$$$$$$$$$$$$$$$$$$$$$$$$$$$$$$$$$ Develop Clamp and Unclamp Interlocks $$$$$$$$$$$$$$$$$$$$$$*)
(* Note: This is one method to create valve bank commands for clamp and unclamp sequencing
you are welcome to use the direct method as well*)

	(*Start Clamp Sequence*)
	(*First Stage Clamping*)
	Clamp_Step.0:= Auto_Run AND NOT Welding_Complete AND FALSE;
	(*Second Stage Clamping*)
	Clamp_Step.1:=  Clamp_Step.0 AND FALSE;
	(*Third Stage Clamping*)
	Clamp_Step.2:= Clamp_Step.1 AND FALSE;
	(*Forth Stage Clamping*)
	Clamp_Step.3:= Clamp_Step.2 AND FALSE;


	(*Start Unlcamp Sequence*)
	(*First Stage Unclamping*)
	Unclamp_Step.0:= Welding_Complete AND FALSE;
	(*Second Stage Unclamping*)
	Unclamp_Step.1:= Unclamp_Step.0 AND FALSE;
	(*Third Stage Unclamping*)
	Unclamp_Step.2:= Unclamp_Step.1 AND FALSE;
	(*Fourth Stage Unclamping*)
	Unclamp_Step.3:= Unclamp_Step.2 AND FALSE;



(*------------------------------------------- Repositions --------------------------------------*)

	(*Reposition Request#1*)
	IF FALSE
		THEN
			Repo_Reqs.0:= TRUE;
	END_IF;

	(*Reposition Request#2*)
	IF FALSE
		THEN
			Repo_Reqs.1:= TRUE;
	END_IF;

	(*Reposition Request#3*)
	IF FALSE
		THEN
			Repo_Reqs.2:= TRUE;
	END_IF;

	(*Reposition Request#4*)
	IF FALSE
		THEN
			Repo_Reqs.3:= TRUE;
	END_IF;

	(*Reposition Request#5*)
	IF FALSE
		THEN
			Repo_Reqs.4:= TRUE;
	END_IF;

	(*Reposition Request#6*)
	IF FALSE
		THEN
			Repo_Reqs.5:= TRUE;
	END_IF;

	(*Reposition Request#7*)
	IF FALSE
		THEN
			Repo_Reqs.6:= TRUE;
	END_IF;

	(*Reposition Request#8*)
	IF FALSE
		THEN
			Repo_Reqs.7:= TRUE;
	END_IF;

	(*Reset All Reposition Acks At the End Of Cycle*)
	IF Cycle_Complete
		THEN
			Repo_Reqs:= 0;
	END_IF;

(*------------------------- Reposition Acks ---------------------*)
	Repo_Ack.0:= Repo_Reqs.0 AND FALSE;
	Repo_Ack.1:= Repo_Reqs.1 AND FALSE;
	Repo_Ack.2:= Repo_Reqs.2 AND FALSE;
	Repo_Ack.3:= Repo_Reqs.3 AND FALSE;
	Repo_Ack.4:= Repo_Reqs.4 AND FALSE;
	Repo_Ack.5:= Repo_Reqs.5 AND FALSE;
	Repo_Ack.6:= Repo_Reqs.6 AND FALSE;
	Repo_Ack.7:= Repo_Reqs.7 AND FALSE;
END_ACTION

ACTION ValveBank1:


(*+++++++++++THIS AREA IS CUSTOM PER INSTALLATION AND WILL HAVE TO BE MODIFIED PER +++++++++++++*)
(*+++++++++++THIS AREA IS CUSTOM PER INSTALLATION AND WILL HAVE TO BE MODIFIED PER +++++++++++++*)
(*+++++++++++THIS AREA IS CUSTOM PER INSTALLATION AND WILL HAVE TO BE MODIFIED PER +++++++++++++*)

(*+++++++++++VALVE BANK 1 +++++++++++++*)
(*+++++++++++VALVE BANK 1 +++++++++++++*)
(*+++++++++++VALVE BANK 1 +++++++++++++*)


	(*Valve 1, A+B*)
	(*spare*)
		Valve1FB
			(
			Enable_Motion:= Enable_Motion ,
			Enable_Latch:= TRUE,					(*Enabling Runs Valve as detent type (maintained solenoids*)
			Enable_SideA_PreCharge:= FALSE,		(*Enabling Turns Side A PreCharge Active, reset when Side B is energized in Auto*)
			Enable_SideB_PreCharge:= FALSE,		(*Enabling Turns Side B PreCharge Active, reset when Side A is energized in Auto*)
			PreCharge_Time:= T#0.1S,
			Enable_Auto_Commands:= In_Auto,
			Enable_Manual_Commands:= In_Manual AND All_Robots_Clear,
			In_Manual_SideA_Command:= Discrete_In.ManReqs.0,
			In_Manual_SideB_Command:= (Discrete_In.ManReqs.1 OR Discrete_In.Go_Home),
			SideA_Indicator:= (Clamp1ADVD AND Clamp2ADVD AND Clamp3ADVD AND Clamp4ADVD),
			SideB_Indicator:= (Clamp1RETD AND Clamp2RETD AND Clamp3RETD AND Clamp4RETD) OR Manual_Ind_HomePrompt,
			TurnOn_SideA_SOL=> N100.Q.0,
			TurnOn_SideB_SOL=> N100.Q.1,
			TurnOn_SideA_Indicator=> Manual_Indicators1.0,
			TurnOn_SideB_Indicator=> Manual_Indicators1.1
			 );
		Valve1FB.In_Auto_SideA_Command:= FALSE;
		Valve1FB.In_Auto_SideB_Command:= FALSE;


	(*Valve 2, A+B*)
	(*spare*)
		Valve2FB
			(
			Enable_Motion:= Enable_Motion ,
			Enable_Latch:= TRUE,					(*Enabling Runs Valve as detent type (maintained solenoids*)
			Enable_SideA_PreCharge:= FALSE,		(*Enabling Turns Side A PreCharge Active, reset when Side B is energized in Auto*)
			Enable_SideB_PreCharge:= FALSE,		(*Enabling Turns Side B PreCharge Active, reset when Side A is energized in Auto*)
			PreCharge_Time:= T#0.10S,
			Enable_Auto_Commands:= In_Auto,
			Enable_Manual_Commands:= In_Manual AND All_Robots_Clear,
			In_Manual_SideA_Command:= Discrete_In.ManReqs.2,
			In_Manual_SideB_Command:= Discrete_In.ManReqs.3,
			SideA_Indicator:= FALSE,
			SideB_Indicator:= FALSE,
			TurnOn_SideA_SOL=> N100.Q.2,
			TurnOn_SideB_SOL=> N100.Q.3,
			TurnOn_SideA_Indicator=> Manual_Indicators1.2,
			TurnOn_SideB_Indicator=> Manual_Indicators1.3
			 );
		Valve2FB.In_Auto_SideA_Command:= FALSE;
		Valve2FB.In_Auto_SideB_Command:= FALSE;


	(*Valve 3, A+B*)
	(*spare*)
		Valve3FB
			(
			Enable_Motion:= Enable_Motion ,
			Enable_Latch:= TRUE,					(*Enabling Runs Valve as detent type (maintained solenoids*)
			Enable_SideA_PreCharge:= FALSE,		(*Enabling Turns Side A PreCharge Active, reset when Side B is energized in Auto*)
			Enable_SideB_PreCharge:= FALSE,		(*Enabling Turns Side B PreCharge Active, reset when Side A is energized in Auto*)
			PreCharge_Time:= T#0.10S,
			Enable_Auto_Commands:= In_Auto,
			Enable_Manual_Commands:= In_Manual AND All_Robots_Clear,
			In_Manual_SideA_Command:= Discrete_In.ManReqs.4,
			In_Manual_SideB_Command:= Discrete_In.ManReqs.5,
			SideA_Indicator:= FALSE,
			SideB_Indicator:= FALSE,
			TurnOn_SideA_SOL=> N100.Q.4,
			TurnOn_SideB_SOL=> N100.Q.5,
			TurnOn_SideA_Indicator=> Manual_Indicators1.4,
			TurnOn_SideB_Indicator=> Manual_Indicators1.5
			 );
		Valve3FB.In_Auto_SideA_Command:= FALSE;
		Valve3FB.In_Auto_SideB_Command:= FALSE;


	(*Valve 4, A+B*)
	(*spare*)
		Valve4FB
			(
			Enable_Motion:= Enable_Motion ,
			Enable_Latch:= TRUE,					(*Enabling Runs Valve as detent type (maintained solenoids*)
			Enable_SideA_PreCharge:= FALSE,		(*Enabling Turns Side A PreCharge Active, reset when Side B is energized in Auto*)
			Enable_SideB_PreCharge:= FALSE,		(*Enabling Turns Side B PreCharge Active, reset when Side A is energized in Auto*)
			PreCharge_Time:= T#0.10S,
			Enable_Auto_Commands:= In_Auto,
			Enable_Manual_Commands:= In_Manual AND All_Robots_Clear,
			In_Manual_SideA_Command:= Discrete_In.ManReqs.6,
			In_Manual_SideB_Command:= Discrete_In.ManReqs.7,
			SideA_Indicator:= FALSE,
			SideB_Indicator:= FALSE,
			TurnOn_SideA_SOL=> N100.Q.6,
			TurnOn_SideB_SOL=> N100.Q.7,
			TurnOn_SideA_Indicator=> Manual_Indicators1.6,
			TurnOn_SideB_Indicator=> Manual_Indicators1.7
			 );
		Valve4FB.In_Auto_SideA_Command:= FALSE;
		Valve4FB.In_Auto_SideB_Command:= FALSE;


	(*Valve 5, A+B*)
	(*spare*)
		Valve5FB
			(
			Enable_Motion:= Enable_Motion ,
			Enable_Latch:= TRUE,					(*Enabling Runs Valve as detent type (maintained solenoids*)
			Enable_SideA_PreCharge:= FALSE,		(*Enabling Turns Side A PreCharge Active, reset when Side B is energized in Auto*)
			Enable_SideB_PreCharge:= FALSE,		(*Enabling Turns Side B PreCharge Active, reset when Side A is energized in Auto*)
			PreCharge_Time:= T#0.10S,
			Enable_Auto_Commands:= In_Auto,
			Enable_Manual_Commands:= In_Manual AND All_Robots_Clear,
			In_Manual_SideA_Command:= Discrete_In.ManReqs.8,
			In_Manual_SideB_Command:= Discrete_In.ManReqs.9,
			SideA_Indicator:= FALSE,
			SideB_Indicator:= FALSE,
			TurnOn_SideA_SOL=> N100.Q.8,
			TurnOn_SideB_SOL=> N100.Q.9,
			TurnOn_SideA_Indicator=> Manual_Indicators1.8,
			TurnOn_SideB_Indicator=> Manual_Indicators1.9
			 );
		Valve5FB.In_Auto_SideA_Command:= FALSE;
		Valve5FB.In_Auto_SideB_Command:= FALSE;


	(*Valve 6, A+B*)
	(*spare*)
		Valve6FB
			(
			Enable_Motion:= Enable_Motion ,
			Enable_Latch:= TRUE,					(*Enabling Runs Valve as detent type (maintained solenoids*)
			Enable_SideA_PreCharge:= FALSE,		(*Enabling Turns Side A PreCharge Active, reset when Side B is energized in Auto*)
			Enable_SideB_PreCharge:= FALSE,		(*Enabling Turns Side B PreCharge Active, reset when Side A is energized in Auto*)
			PreCharge_Time:= T#0.10S,
			Enable_Auto_Commands:= In_Auto,
			Enable_Manual_Commands:= In_Manual AND All_Robots_Clear,
			In_Manual_SideA_Command:= Discrete_In.ManReqs.10,
			In_Manual_SideB_Command:= Discrete_In.ManReqs.11,
			SideA_Indicator:= FALSE,
			SideB_Indicator:= FALSE,
			TurnOn_SideA_SOL=> N100.Q.10,
			TurnOn_SideB_SOL=> N100.Q.11,
			TurnOn_SideA_Indicator=> Manual_Indicators1.10,
			TurnOn_SideB_Indicator=> Manual_Indicators1.11
			 );
		Valve6FB.In_Auto_SideA_Command:= FALSE;
		Valve6FB.In_Auto_SideB_Command:= FALSE;


	(*Valve 7, A+B*)
	(*spare*)
		Valve7FB
			(
			Enable_Motion:= Enable_Motion ,
			Enable_Latch:= TRUE,					(*Enabling Runs Valve as detent type (maintained solenoids*)
			Enable_SideA_PreCharge:= FALSE,		(*Enabling Turns Side A PreCharge Active, reset when Side B is energized in Auto*)
			Enable_SideB_PreCharge:= FALSE,		(*Enabling Turns Side B PreCharge Active, reset when Side A is energized in Auto*)
			PreCharge_Time:= T#0.10S,
			Enable_Auto_Commands:= In_Auto,
			Enable_Manual_Commands:= In_Manual AND All_Robots_Clear,
			In_Manual_SideA_Command:= Discrete_In.ManReqs.12,
			In_Manual_SideB_Command:= Discrete_In.ManReqs.13,
			SideA_Indicator:= FALSE,
			SideB_Indicator:= FALSE,
			TurnOn_SideA_SOL=> N100.Q.12,
			TurnOn_SideB_SOL=> N100.Q.13,
			TurnOn_SideA_Indicator=> Manual_Indicators1.12,
			TurnOn_SideB_Indicator=> Manual_Indicators1.13
			 );
		Valve7FB.In_Auto_SideA_Command:= FALSE;
		Valve7FB.In_Auto_SideB_Command:= FALSE;


	(*Valve 8, A+B*)
	(*spare*)
		Valve8FB
			(
			Enable_Motion:= Enable_Motion ,
			Enable_Latch:= TRUE,					(*Enabling Runs Valve as detent type (maintained solenoids*)
			Enable_SideA_PreCharge:= FALSE,		(*Enabling Turns Side A PreCharge Active, reset when Side B is energized in Auto*)
			Enable_SideB_PreCharge:= FALSE,		(*Enabling Turns Side B PreCharge Active, reset when Side A is energized in Auto*)
			PreCharge_Time:= T#0.10S,
			Enable_Auto_Commands:= In_Auto,
			Enable_Manual_Commands:= In_Manual AND All_Robots_Clear,
			In_Manual_SideA_Command:= Discrete_In.ManReqs.14,
			In_Manual_SideB_Command:= Discrete_In.ManReqs.15,
			SideA_Indicator:= FALSE,
			SideB_Indicator:= FALSE,
			TurnOn_SideA_SOL=> N100.Q.14,
			TurnOn_SideB_SOL=> N100.Q.15,
			TurnOn_SideA_Indicator=> Manual_Indicators1.14,
			TurnOn_SideB_Indicator=> Manual_Indicators1.15
			 );
		Valve8FB.In_Auto_SideA_Command:= FALSE;
		Valve8FB.In_Auto_SideB_Command:= FALSE;


	(*Valve 9, A+B*)
	(*spare*)
		Valve9FB
			(
			Enable_Motion:= Enable_Motion ,
			Enable_Latch:= TRUE,					(*Enabling Runs Valve as detent type (maintained solenoids*)
			Enable_SideA_PreCharge:= FALSE,		(*Enabling Turns Side A PreCharge Active, reset when Side B is energized in Auto*)
			Enable_SideB_PreCharge:= FALSE,		(*Enabling Turns Side B PreCharge Active, reset when Side A is energized in Auto*)
			PreCharge_Time:= T#0.10S,
			Enable_Auto_Commands:= In_Auto,
			Enable_Manual_Commands:= In_Manual AND All_Robots_Clear,
			In_Manual_SideA_Command:= Discrete_In.ManReqs.16,
			In_Manual_SideB_Command:= Discrete_In.ManReqs.17,
			SideA_Indicator:= FALSE,
			SideB_Indicator:= FALSE,
			TurnOn_SideA_SOL=> N100.Q.16,
			TurnOn_SideB_SOL=> N100.Q.17,
			TurnOn_SideA_Indicator=> Manual_Indicators1.16,
			TurnOn_SideB_Indicator=> Manual_Indicators1.17
			 );
		Valve9FB.In_Auto_SideA_Command:= FALSE;
		Valve9FB.In_Auto_SideB_Command:= FALSE;


	(*Valve 10, A+B*)
	(*spare*)
		Valve10FB
			(
			Enable_Motion:= Enable_Motion ,
			Enable_Latch:= TRUE,					(*Enabling Runs Valve as detent type (maintained solenoids*)
			Enable_SideA_PreCharge:= FALSE,		(*Enabling Turns Side A PreCharge Active, reset when Side B is energized in Auto*)
			Enable_SideB_PreCharge:= FALSE,		(*Enabling Turns Side B PreCharge Active, reset when Side A is energized in Auto*)
			PreCharge_Time:= T#0.10S,
			Enable_Auto_Commands:= In_Auto,
			Enable_Manual_Commands:= In_Manual AND All_Robots_Clear,
			In_Manual_SideA_Command:= Discrete_In.ManReqs.18,
			In_Manual_SideB_Command:= Discrete_In.ManReqs.19,
			SideA_Indicator:= FALSE,
			SideB_Indicator:= FALSE,
			TurnOn_SideA_SOL=> N100.Q.18,
			TurnOn_SideB_SOL=> N100.Q.19,
			TurnOn_SideA_Indicator=> Manual_Indicators1.18,
			TurnOn_SideB_Indicator=> Manual_Indicators1.19
			 );
		Valve10FB.In_Auto_SideA_Command:= FALSE;
		Valve10FB.In_Auto_SideB_Command:= FALSE;


	(*Valve 11, A+B*)
	(*spare*)
		Valve11FB
			(
			Enable_Motion:= Enable_Motion ,
			Enable_Latch:= TRUE,					(*Enabling Runs Valve as detent type (maintained solenoids*)
			Enable_SideA_PreCharge:= FALSE,		(*Enabling Turns Side A PreCharge Active, reset when Side B is energized in Auto*)
			Enable_SideB_PreCharge:= FALSE,		(*Enabling Turns Side B PreCharge Active, reset when Side A is energized in Auto*)
			PreCharge_Time:= T#0.10S,
			Enable_Auto_Commands:= In_Auto,
			Enable_Manual_Commands:= In_Manual AND All_Robots_Clear,
			In_Manual_SideA_Command:= Discrete_In.ManReqs.20,
			In_Manual_SideB_Command:= Discrete_In.ManReqs.21,
			SideA_Indicator:= FALSE,
			SideB_Indicator:= FALSE,
			TurnOn_SideA_SOL=> N100.Q.20,
			TurnOn_SideB_SOL=> N100.Q.21,
			TurnOn_SideA_Indicator=> Manual_Indicators1.20,
			TurnOn_SideB_Indicator=> Manual_Indicators1.21
			 );
		Valve11FB.In_Auto_SideA_Command:= FALSE;
		Valve11FB.In_Auto_SideB_Command:= FALSE;


	(*Valve 12, A+B*)
	(*spare*)
		Valve12FB
			(
			Enable_Motion:= Enable_Motion ,
			Enable_Latch:= TRUE,					(*Enabling Runs Valve as detent type (maintained solenoids*)
			Enable_SideA_PreCharge:= FALSE,		(*Enabling Turns Side A PreCharge Active, reset when Side B is energized in Auto*)
			Enable_SideB_PreCharge:= FALSE,		(*Enabling Turns Side B PreCharge Active, reset when Side A is energized in Auto*)
			PreCharge_Time:= T#0.10S,
			Enable_Auto_Commands:= In_Auto,
			Enable_Manual_Commands:= In_Manual AND All_Robots_Clear,
			In_Manual_SideA_Command:= Discrete_In.ManReqs.22,
			In_Manual_SideB_Command:= Discrete_In.ManReqs.23,
			SideA_Indicator:= FALSE,
			SideB_Indicator:= FALSE,
			TurnOn_SideA_SOL=> N100.Q.22,
			TurnOn_SideB_SOL=> N100.Q.23,
			TurnOn_SideA_Indicator=> Manual_Indicators1.22,
			TurnOn_SideB_Indicator=> Manual_Indicators1.23
			 );
		Valve12FB.In_Auto_SideA_Command:= FALSE;
		Valve12FB.In_Auto_SideB_Command:= FALSE;


	(*Valve 13, A+B*)
	(*spare*)
		Valve13FB
			(
			Enable_Motion:= Enable_Motion ,
			Enable_Latch:= TRUE,					(*Enabling Runs Valve as detent type (maintained solenoids*)
			Enable_SideA_PreCharge:= FALSE,		(*Enabling Turns Side A PreCharge Active, reset when Side B is energized in Auto*)
			Enable_SideB_PreCharge:= FALSE,		(*Enabling Turns Side B PreCharge Active, reset when Side A is energized in Auto*)
			PreCharge_Time:= T#0.10S,
			Enable_Auto_Commands:= In_Auto,
			Enable_Manual_Commands:= In_Manual AND All_Robots_Clear,
			In_Manual_SideA_Command:= Discrete_In.ManReqs.24,
			In_Manual_SideB_Command:= Discrete_In.ManReqs.25,
			SideA_Indicator:= FALSE,
			SideB_Indicator:= FALSE,
			TurnOn_SideA_SOL=> N100.Q.24,
			TurnOn_SideB_SOL=> N100.Q.25,
			TurnOn_SideA_Indicator=> Manual_Indicators1.24,
			TurnOn_SideB_Indicator=> Manual_Indicators1.25
			 );
		Valve13FB.In_Auto_SideA_Command:= FALSE;
		Valve13FB.In_Auto_SideB_Command:= FALSE;


	(*Valve 14, A+B*)
	(*spare*)
		Valve14FB
			(
			Enable_Motion:= Enable_Motion ,
			Enable_Latch:= TRUE,					(*Enabling Runs Valve as detent type (maintained solenoids*)
			Enable_SideA_PreCharge:= FALSE,		(*Enabling Turns Side A PreCharge Active, reset when Side B is energized in Auto*)
			Enable_SideB_PreCharge:= FALSE,		(*Enabling Turns Side B PreCharge Active, reset when Side A is energized in Auto*)
			PreCharge_Time:= T#0.10S,
			Enable_Auto_Commands:= In_Auto,
			Enable_Manual_Commands:= In_Manual AND All_Robots_Clear,
			In_Manual_SideA_Command:= Discrete_In.ManReqs.26,
			In_Manual_SideB_Command:= Discrete_In.ManReqs.27,
			SideA_Indicator:= FALSE,
			SideB_Indicator:= FALSE,
			TurnOn_SideA_SOL=> N100.Q.26,
			TurnOn_SideB_SOL=> N100.Q.27,
			TurnOn_SideA_Indicator=> Manual_Indicators1.26,
			TurnOn_SideB_Indicator=> Manual_Indicators1.27
			 );
		Valve14FB.In_Auto_SideA_Command:= FALSE;
		Valve14FB.In_Auto_SideB_Command:= FALSE;


	(*Valve 15, A+B*)
	(*spare*)
		Valve15FB
			(
			Enable_Motion:= Enable_Motion ,
			Enable_Latch:= TRUE,					(*Enabling Runs Valve as detent type (maintained solenoids*)
			Enable_SideA_PreCharge:= FALSE,		(*Enabling Turns Side A PreCharge Active, reset when Side B is energized in Auto*)
			Enable_SideB_PreCharge:= FALSE,		(*Enabling Turns Side B PreCharge Active, reset when Side A is energized in Auto*)
			PreCharge_Time:= T#0.10S,
			Enable_Auto_Commands:= In_Auto,
			Enable_Manual_Commands:= In_Manual AND All_Robots_Clear,
			In_Manual_SideA_Command:= Discrete_In.ManReqs.28,
			In_Manual_SideB_Command:= Discrete_In.ManReqs.29,
			SideA_Indicator:= FALSE,
			SideB_Indicator:= FALSE,
			TurnOn_SideA_SOL=> N100.Q.28,
			TurnOn_SideB_SOL=> N100.Q.29,
			TurnOn_SideA_Indicator=> Manual_Indicators1.28,
			TurnOn_SideB_Indicator=> Manual_Indicators1.29
			 );
		Valve15FB.In_Auto_SideA_Command:= FALSE;
		Valve15FB.In_Auto_SideB_Command:= FALSE;


	(*Valve 16, A+B*)
	(*spare*)
		Valve16FB
			(
			Enable_Motion:= Enable_Motion ,
			Enable_Latch:= TRUE,					(*Enabling Runs Valve as detent type (maintained solenoids*)
			Enable_SideA_PreCharge:= FALSE,		(*Enabling Turns Side A PreCharge Active, reset when Side B is energized in Auto*)
			Enable_SideB_PreCharge:= FALSE,		(*Enabling Turns Side B PreCharge Active, reset when Side A is energized in Auto*)
			PreCharge_Time:= T#0.10S,
			Enable_Auto_Commands:= In_Auto,
			Enable_Manual_Commands:= In_Manual AND All_Robots_Clear,
			In_Manual_SideA_Command:= Discrete_In.ManReqs.30,
			In_Manual_SideB_Command:= Discrete_In.ManReqs.31,
			SideA_Indicator:= FALSE,
			SideB_Indicator:= FALSE,
			TurnOn_SideA_SOL=> N100.Q.30,
			TurnOn_SideB_SOL=> N100.Q.31,
			TurnOn_SideA_Indicator=> Manual_Indicators1.30,
			TurnOn_SideB_Indicator=> Manual_Indicators1.31
			 );
		Valve16FB.In_Auto_SideA_Command:= FALSE;
		Valve16FB.In_Auto_SideB_Command:= FALSE;


























(*end*)
END_ACTION

ACTION ValveBank2:


(*+++++++++++THIS AREA IS CUSTOM PER INSTALLATION AND WILL HAVE TO BE MODIFIED PER +++++++++++++*)
(*+++++++++++THIS AREA IS CUSTOM PER INSTALLATION AND WILL HAVE TO BE MODIFIED PER +++++++++++++*)
(*+++++++++++THIS AREA IS CUSTOM PER INSTALLATION AND WILL HAVE TO BE MODIFIED PER +++++++++++++*)

(*+++++++++++VALVE BANK 2 +++++++++++++*)
(*+++++++++++VALVE BANK 2 +++++++++++++*)
(*+++++++++++VALVE BANK 2 +++++++++++++*)


	(*Valve 17, A+B*)
	(*spare*)
		Valve17FB
			(
			Enable_Motion:= Enable_Motion ,
			Enable_Latch:= TRUE,					(*Enabling Runs Valve as detent type (maintained solenoids*)
			Enable_SideA_PreCharge:= FALSE,		(*Enabling Turns Side A PreCharge Active, reset when Side B is energized in Auto*)
			Enable_SideB_PreCharge:= FALSE,		(*Enabling Turns Side B PreCharge Active, reset when Side A is energized in Auto*)
			PreCharge_Time:= T#0.1S,
			Enable_Auto_Commands:= In_Auto,
			Enable_Manual_Commands:= In_Manual AND All_Robots_Clear,
			In_Manual_SideA_Command:= Discrete_In.ManReqs2.0,
			In_Manual_SideB_Command:= (Discrete_In.ManReqs2.1 OR Discrete_In.Go_Home),
			SideA_Indicator:= FALSE,
			SideB_Indicator:= FALSE,
			TurnOn_SideA_SOL=> N101.Q.0,
			TurnOn_SideB_SOL=> N101.Q.1,
			TurnOn_SideA_Indicator=> Manual_Indicators2.0,
			TurnOn_SideB_Indicator=> Manual_Indicators2.1
			 );
		Valve17FB.In_Auto_SideA_Command:= FALSE;
		Valve17FB.In_Auto_SideB_Command:= FALSE;


	(*Valve 18, A+B*)
	(*spare*)
		Valve18FB
			(
			Enable_Motion:= Enable_Motion ,
			Enable_Latch:= TRUE,					(*Enabling Runs Valve as detent type (maintained solenoids*)
			Enable_SideA_PreCharge:= FALSE,		(*Enabling Turns Side A PreCharge Active, reset when Side B is energized in Auto*)
			Enable_SideB_PreCharge:= FALSE,		(*Enabling Turns Side B PreCharge Active, reset when Side A is energized in Auto*)
			PreCharge_Time:= T#0.10S,
			Enable_Auto_Commands:= In_Auto,
			Enable_Manual_Commands:= In_Manual AND All_Robots_Clear,
			In_Manual_SideA_Command:= Discrete_In.ManReqs2.2,
			In_Manual_SideB_Command:= Discrete_In.ManReqs2.3,
			SideA_Indicator:= FALSE,
			SideB_Indicator:= FALSE,
			TurnOn_SideA_SOL=> N101.Q.2,
			TurnOn_SideB_SOL=> N101.Q.3,
			TurnOn_SideA_Indicator=> Manual_Indicators2.2,
			TurnOn_SideB_Indicator=> Manual_Indicators2.3
			 );
		Valve18FB.In_Auto_SideA_Command:= FALSE;
		Valve18FB.In_Auto_SideB_Command:= FALSE;

	(*Valve 19, A+B*)
	(*spare*)
		Valve19FB
			(
			Enable_Motion:= Enable_Motion ,
			Enable_Latch:= TRUE,					(*Enabling Runs Valve as detent type (maintained solenoids*)
			Enable_SideA_PreCharge:= FALSE,		(*Enabling Turns Side A PreCharge Active, reset when Side B is energized in Auto*)
			Enable_SideB_PreCharge:= FALSE,		(*Enabling Turns Side B PreCharge Active, reset when Side A is energized in Auto*)
			PreCharge_Time:= T#0.10S,
			Enable_Auto_Commands:= In_Auto,
			Enable_Manual_Commands:= In_Manual AND All_Robots_Clear,
			In_Manual_SideA_Command:= Discrete_In.ManReqs2.4,
			In_Manual_SideB_Command:= Discrete_In.ManReqs2.5,
			SideA_Indicator:= FALSE,
			SideB_Indicator:= FALSE,
			TurnOn_SideA_SOL=> N101.Q.4,
			TurnOn_SideB_SOL=> N101.Q.5,
			TurnOn_SideA_Indicator=> Manual_Indicators2.4,
			TurnOn_SideB_Indicator=> Manual_Indicators2.5
			 );
		Valve19FB.In_Auto_SideA_Command:= FALSE;
		Valve19FB.In_Auto_SideB_Command:= FALSE;


	(*Valve 20, A+B*)
	(*spare*)
		Valve20FB
			(
			Enable_Motion:= Enable_Motion ,
			Enable_Latch:= TRUE,					(*Enabling Runs Valve as detent type (maintained solenoids*)
			Enable_SideA_PreCharge:= FALSE,		(*Enabling Turns Side A PreCharge Active, reset when Side B is energized in Auto*)
			Enable_SideB_PreCharge:= FALSE,		(*Enabling Turns Side B PreCharge Active, reset when Side A is energized in Auto*)
			PreCharge_Time:= T#0.10S,
			Enable_Auto_Commands:= In_Auto,
			Enable_Manual_Commands:= In_Manual AND All_Robots_Clear,
			In_Manual_SideA_Command:= Discrete_In.ManReqs2.6,
			In_Manual_SideB_Command:= Discrete_In.ManReqs2.7,
			SideA_Indicator:= FALSE,
			SideB_Indicator:= FALSE,
			TurnOn_SideA_SOL=> N101.Q.6,
			TurnOn_SideB_SOL=> N101.Q.7,
			TurnOn_SideA_Indicator=> Manual_Indicators2.6,
			TurnOn_SideB_Indicator=> Manual_Indicators2.7
			 );
		Valve20FB.In_Auto_SideA_Command:= FALSE;
		Valve20FB.In_Auto_SideB_Command:= FALSE;


	(*Valve 21, A+B*)
	(*spare*)
		Valve21FB
			(
			Enable_Motion:= Enable_Motion ,
			Enable_Latch:= TRUE,					(*Enabling Runs Valve as detent type (maintained solenoids*)
			Enable_SideA_PreCharge:= FALSE,		(*Enabling Turns Side A PreCharge Active, reset when Side B is energized in Auto*)
			Enable_SideB_PreCharge:= FALSE,		(*Enabling Turns Side B PreCharge Active, reset when Side A is energized in Auto*)
			PreCharge_Time:= T#0.10S,
			Enable_Auto_Commands:= In_Auto,
			Enable_Manual_Commands:= In_Manual AND All_Robots_Clear,
			In_Manual_SideA_Command:= Discrete_In.ManReqs2.8,
			In_Manual_SideB_Command:= Discrete_In.ManReqs2.9,
			SideA_Indicator:= FALSE,
			SideB_Indicator:= FALSE,
			TurnOn_SideA_SOL=> N101.Q.8,
			TurnOn_SideB_SOL=> N101.Q.9,
			TurnOn_SideA_Indicator=> Manual_Indicators2.8,
			TurnOn_SideB_Indicator=> Manual_Indicators2.9
			 );
		Valve21FB.In_Auto_SideA_Command:= FALSE;
		Valve21FB.In_Auto_SideB_Command:= FALSE;


	(*Valve 22, A+B*)
	(*spare*)
		Valve22FB
			(
			Enable_Motion:= Enable_Motion ,
			Enable_Latch:= TRUE,					(*Enabling Runs Valve as detent type (maintained solenoids*)
			Enable_SideA_PreCharge:= FALSE,		(*Enabling Turns Side A PreCharge Active, reset when Side B is energized in Auto*)
			Enable_SideB_PreCharge:= FALSE,		(*Enabling Turns Side B PreCharge Active, reset when Side A is energized in Auto*)
			PreCharge_Time:= T#0.10S,
			Enable_Auto_Commands:= In_Auto,
			Enable_Manual_Commands:= In_Manual AND All_Robots_Clear,
			In_Manual_SideA_Command:= Discrete_In.ManReqs2.10,
			In_Manual_SideB_Command:= Discrete_In.ManReqs2.11,
			SideA_Indicator:= FALSE,
			SideB_Indicator:= FALSE,
			TurnOn_SideA_SOL=> N101.Q.10,
			TurnOn_SideB_SOL=> N101.Q.11,
			TurnOn_SideA_Indicator=> Manual_Indicators2.10,
			TurnOn_SideB_Indicator=> Manual_Indicators2.11
			 );
		Valve22FB.In_Auto_SideA_Command:= FALSE;
		Valve22FB.In_Auto_SideB_Command:= FALSE;


	(*Valve 23, A+B*)
	(*spare*)
		Valve23FB
			(
			Enable_Motion:= Enable_Motion ,
			Enable_Latch:= TRUE,					(*Enabling Runs Valve as detent type (maintained solenoids*)
			Enable_SideA_PreCharge:= FALSE,		(*Enabling Turns Side A PreCharge Active, reset when Side B is energized in Auto*)
			Enable_SideB_PreCharge:= FALSE,		(*Enabling Turns Side B PreCharge Active, reset when Side A is energized in Auto*)
			PreCharge_Time:= T#0.10S,
			Enable_Auto_Commands:= In_Auto,
			Enable_Manual_Commands:= In_Manual AND All_Robots_Clear,
			In_Manual_SideA_Command:= Discrete_In.ManReqs2.12,
			In_Manual_SideB_Command:= Discrete_In.ManReqs2.13,
			SideA_Indicator:= FALSE,
			SideB_Indicator:= FALSE,
			TurnOn_SideA_SOL=> N101.Q.12,
			TurnOn_SideB_SOL=> N101.Q.13,
			TurnOn_SideA_Indicator=> Manual_Indicators2.12,
			TurnOn_SideB_Indicator=> Manual_Indicators2.13
			 );
		Valve23FB.In_Auto_SideA_Command:= FALSE;
		Valve23FB.In_Auto_SideB_Command:= FALSE;


	(*Valve 24, A+B*)
	(*spare*)
		Valve24FB
			(
			Enable_Motion:= Enable_Motion ,
			Enable_Latch:= TRUE,					(*Enabling Runs Valve as detent type (maintained solenoids*)
			Enable_SideA_PreCharge:= FALSE,		(*Enabling Turns Side A PreCharge Active, reset when Side B is energized in Auto*)
			Enable_SideB_PreCharge:= FALSE,		(*Enabling Turns Side B PreCharge Active, reset when Side A is energized in Auto*)
			PreCharge_Time:= T#0.10S,
			Enable_Auto_Commands:= In_Auto,
			Enable_Manual_Commands:= In_Manual AND All_Robots_Clear,
			In_Manual_SideA_Command:= Discrete_In.ManReqs2.14,
			In_Manual_SideB_Command:= Discrete_In.ManReqs2.15,
			SideA_Indicator:= FALSE,
			SideB_Indicator:= FALSE,
			TurnOn_SideA_SOL=> N101.Q.14,
			TurnOn_SideB_SOL=> N101.Q.15,
			TurnOn_SideA_Indicator=> Manual_Indicators2.14,
			TurnOn_SideB_Indicator=> Manual_Indicators2.15
			 );
		Valve24FB.In_Auto_SideA_Command:= FALSE;
		Valve24FB.In_Auto_SideB_Command:= FALSE;


	(*Valve 25, A+B*)
	(*spare*)
		Valve25FB
			(
			Enable_Motion:= Enable_Motion ,
			Enable_Latch:= TRUE,					(*Enabling Runs Valve as detent type (maintained solenoids*)
			Enable_SideA_PreCharge:= FALSE,		(*Enabling Turns Side A PreCharge Active, reset when Side B is energized in Auto*)
			Enable_SideB_PreCharge:= FALSE,		(*Enabling Turns Side B PreCharge Active, reset when Side A is energized in Auto*)
			PreCharge_Time:= T#0.10S,
			Enable_Auto_Commands:= In_Auto,
			Enable_Manual_Commands:= In_Manual AND All_Robots_Clear,
			In_Manual_SideA_Command:= Discrete_In.ManReqs2.16,
			In_Manual_SideB_Command:= Discrete_In.ManReqs2.17,
			SideA_Indicator:= FALSE,
			SideB_Indicator:= FALSE,
			TurnOn_SideA_SOL=> N101.Q.16,
			TurnOn_SideB_SOL=> N101.Q.17,
			TurnOn_SideA_Indicator=> Manual_Indicators2.16,
			TurnOn_SideB_Indicator=> Manual_Indicators2.17
			 );
		Valve25FB.In_Auto_SideA_Command:= FALSE;
		Valve25FB.In_Auto_SideB_Command:= FALSE;


	(*Valve 26, A+B*)
	(*spare*)
		Valve26FB
			(
			Enable_Motion:= Enable_Motion ,
			Enable_Latch:= TRUE,					(*Enabling Runs Valve as detent type (maintained solenoids*)
			Enable_SideA_PreCharge:= FALSE,		(*Enabling Turns Side A PreCharge Active, reset when Side B is energized in Auto*)
			Enable_SideB_PreCharge:= FALSE,		(*Enabling Turns Side B PreCharge Active, reset when Side A is energized in Auto*)
			PreCharge_Time:= T#0.10S,
			Enable_Auto_Commands:= In_Auto,
			Enable_Manual_Commands:= In_Manual AND All_Robots_Clear,
			In_Manual_SideA_Command:= Discrete_In.ManReqs2.18,
			In_Manual_SideB_Command:= Discrete_In.ManReqs2.19,
			SideA_Indicator:= FALSE,
			SideB_Indicator:= FALSE,
			TurnOn_SideA_SOL=> N101.Q.18,
			TurnOn_SideB_SOL=> N101.Q.19,
			TurnOn_SideA_Indicator=> Manual_Indicators2.18,
			TurnOn_SideB_Indicator=> Manual_Indicators2.19
			 );
		Valve26FB.In_Auto_SideA_Command:= FALSE;
		Valve26FB.In_Auto_SideB_Command:= FALSE;


	(*Valve 27, A+B*)
	(*spare*)
		Valve27FB
			(
			Enable_Motion:= Enable_Motion ,
			Enable_Latch:= TRUE,					(*Enabling Runs Valve as detent type (maintained solenoids*)
			Enable_SideA_PreCharge:= FALSE,		(*Enabling Turns Side A PreCharge Active, reset when Side B is energized in Auto*)
			Enable_SideB_PreCharge:= FALSE,		(*Enabling Turns Side B PreCharge Active, reset when Side A is energized in Auto*)
			PreCharge_Time:= T#0.10S,
			Enable_Auto_Commands:= In_Auto,
			Enable_Manual_Commands:= In_Manual AND All_Robots_Clear,
			In_Manual_SideA_Command:= Discrete_In.ManReqs2.20,
			In_Manual_SideB_Command:= Discrete_In.ManReqs2.21,
			SideA_Indicator:= FALSE,
			SideB_Indicator:= FALSE,
			TurnOn_SideA_SOL=> N101.Q.20,
			TurnOn_SideB_SOL=> N101.Q.21,
			TurnOn_SideA_Indicator=> Manual_Indicators2.20,
			TurnOn_SideB_Indicator=> Manual_Indicators2.21
			 );
		Valve27FB.In_Auto_SideA_Command:= FALSE;
		Valve27FB.In_Auto_SideB_Command:= FALSE;


	(*Valve 28, A+B*)
	(*spare*)
		Valve28FB
			(
			Enable_Motion:= Enable_Motion ,
			Enable_Latch:= TRUE,					(*Enabling Runs Valve as detent type (maintained solenoids*)
			Enable_SideA_PreCharge:= FALSE,		(*Enabling Turns Side A PreCharge Active, reset when Side B is energized in Auto*)
			Enable_SideB_PreCharge:= FALSE,		(*Enabling Turns Side B PreCharge Active, reset when Side A is energized in Auto*)
			PreCharge_Time:= T#0.10S,
			Enable_Auto_Commands:= In_Auto,
			Enable_Manual_Commands:= In_Manual AND All_Robots_Clear,
			In_Manual_SideA_Command:= Discrete_In.ManReqs2.22,
			In_Manual_SideB_Command:= Discrete_In.ManReqs2.23,
			SideA_Indicator:= FALSE,
			SideB_Indicator:= FALSE,
			TurnOn_SideA_SOL=> N101.Q.22,
			TurnOn_SideB_SOL=> N101.Q.23,
			TurnOn_SideA_Indicator=> Manual_Indicators2.22,
			TurnOn_SideB_Indicator=> Manual_Indicators2.23
			 );
		Valve28FB.In_Auto_SideA_Command:= FALSE;
		Valve28FB.In_Auto_SideB_Command:= FALSE;


	(*Valve 29, A+B*)
	(*spare*)
		Valve29FB
			(
			Enable_Motion:= Enable_Motion ,
			Enable_Latch:= TRUE,					(*Enabling Runs Valve as detent type (maintained solenoids*)
			Enable_SideA_PreCharge:= FALSE,		(*Enabling Turns Side A PreCharge Active, reset when Side B is energized in Auto*)
			Enable_SideB_PreCharge:= FALSE,		(*Enabling Turns Side B PreCharge Active, reset when Side A is energized in Auto*)
			PreCharge_Time:= T#0.10S,
			Enable_Auto_Commands:= In_Auto,
			Enable_Manual_Commands:= In_Manual AND All_Robots_Clear,
			In_Manual_SideA_Command:= Discrete_In.ManReqs2.24,
			In_Manual_SideB_Command:= Discrete_In.ManReqs2.25,
			SideA_Indicator:= FALSE,
			SideB_Indicator:= FALSE,
			TurnOn_SideA_SOL=> N101.Q.24,
			TurnOn_SideB_SOL=> N101.Q.25,
			TurnOn_SideA_Indicator=> Manual_Indicators2.24,
			TurnOn_SideB_Indicator=> Manual_Indicators2.25
			 );
		Valve29FB.In_Auto_SideA_Command:= FALSE;
		Valve29FB.In_Auto_SideB_Command:= FALSE;


	(*Valve 30, A+B*)
	(*spare*)
		Valve30FB
			(
			Enable_Motion:= Enable_Motion ,
			Enable_Latch:= TRUE,					(*Enabling Runs Valve as detent type (maintained solenoids*)
			Enable_SideA_PreCharge:= FALSE,		(*Enabling Turns Side A PreCharge Active, reset when Side B is energized in Auto*)
			Enable_SideB_PreCharge:= FALSE,		(*Enabling Turns Side B PreCharge Active, reset when Side A is energized in Auto*)
			PreCharge_Time:= T#0.10S,
			Enable_Auto_Commands:= In_Auto,
			Enable_Manual_Commands:= In_Manual AND All_Robots_Clear,
			In_Manual_SideA_Command:= Discrete_In.ManReqs2.26,
			In_Manual_SideB_Command:= Discrete_In.ManReqs2.27,
			SideA_Indicator:= FALSE,
			SideB_Indicator:= FALSE,
			TurnOn_SideA_SOL=> N101.Q.26,
			TurnOn_SideB_SOL=> N101.Q.27,
			TurnOn_SideA_Indicator=> Manual_Indicators2.26,
			TurnOn_SideB_Indicator=> Manual_Indicators2.27
			 );
		Valve30FB.In_Auto_SideA_Command:= FALSE;
		Valve30FB.In_Auto_SideB_Command:= FALSE;


	(*Valve 31, A+B*)
	(*spare*)
		Valve31FB
			(
			Enable_Motion:= Enable_Motion ,
			Enable_Latch:= TRUE,					(*Enabling Runs Valve as detent type (maintained solenoids*)
			Enable_SideA_PreCharge:= FALSE,		(*Enabling Turns Side A PreCharge Active, reset when Side B is energized in Auto*)
			Enable_SideB_PreCharge:= FALSE,		(*Enabling Turns Side B PreCharge Active, reset when Side A is energized in Auto*)
			PreCharge_Time:= T#0.10S,
			Enable_Auto_Commands:= In_Auto,
			Enable_Manual_Commands:= In_Manual AND All_Robots_Clear,
			In_Manual_SideA_Command:= Discrete_In.ManReqs2.28,
			In_Manual_SideB_Command:= Discrete_In.ManReqs2.29,
			SideA_Indicator:= FALSE,
			SideB_Indicator:= FALSE,
			TurnOn_SideA_SOL=> N101.Q.28,
			TurnOn_SideB_SOL=> N101.Q.29,
			TurnOn_SideA_Indicator=> Manual_Indicators2.28,
			TurnOn_SideB_Indicator=> Manual_Indicators2.29
			 );
		Valve31FB.In_Auto_SideA_Command:= FALSE;
		Valve31FB.In_Auto_SideB_Command:= FALSE;


	(*Valve 32, A+B*)
	(*spare*)
		Valve32FB
			(
			Enable_Motion:= Enable_Motion ,
			Enable_Latch:= TRUE,					(*Enabling Runs Valve as detent type (maintained solenoids*)
			Enable_SideA_PreCharge:= FALSE,		(*Enabling Turns Side A PreCharge Active, reset when Side B is energized in Auto*)
			Enable_SideB_PreCharge:= FALSE,		(*Enabling Turns Side B PreCharge Active, reset when Side A is energized in Auto*)
			PreCharge_Time:= T#0.10S,
			Enable_Auto_Commands:= In_Auto,
			Enable_Manual_Commands:= In_Manual AND All_Robots_Clear,
			In_Manual_SideA_Command:= Discrete_In.ManReqs2.30,
			In_Manual_SideB_Command:= Discrete_In.ManReqs2.31,
			SideA_Indicator:= FALSE,
			SideB_Indicator:= FALSE,
			TurnOn_SideA_SOL=> N101.Q.30,
			TurnOn_SideB_SOL=> N101.Q.31,
			TurnOn_SideA_Indicator=> Manual_Indicators2.30,
			TurnOn_SideB_Indicator=> Manual_Indicators2.31
			 );
		Valve32FB.In_Auto_SideA_Command:= FALSE;
		Valve32FB.In_Auto_SideB_Command:= FALSE;




















(*end*)
END_ACTION

ACTION ValveBank3:


(*+++++++++++THIS AREA IS CUSTOM PER INSTALLATION AND WILL HAVE TO BE MODIFIED PER +++++++++++++*)
(*+++++++++++THIS AREA IS CUSTOM PER INSTALLATION AND WILL HAVE TO BE MODIFIED PER +++++++++++++*)
(*+++++++++++THIS AREA IS CUSTOM PER INSTALLATION AND WILL HAVE TO BE MODIFIED PER +++++++++++++*)

(*+++++++++++VALVE BANK 3 +++++++++++++*)
(*+++++++++++VALVE BANK 3 +++++++++++++*)
(*+++++++++++VALVE BANK 3 +++++++++++++*)


	(*Valve 33, A+B*)
	(*spare*)
		Valve33FB
			(
			Enable_Motion:= Enable_Motion ,
			Enable_Latch:= TRUE,					(*Enabling Runs Valve as detent type (maintained solenoids*)
			Enable_SideA_PreCharge:= FALSE,		(*Enabling Turns Side A PreCharge Active, reset when Side B is energized in Auto*)
			Enable_SideB_PreCharge:= FALSE,		(*Enabling Turns Side B PreCharge Active, reset when Side A is energized in Auto*)
			PreCharge_Time:= T#0.1S,
			Enable_Auto_Commands:= In_Auto,
			Enable_Manual_Commands:= In_Manual AND All_Robots_Clear,
			In_Manual_SideA_Command:= Discrete_In.ManReqs3.0,
			In_Manual_SideB_Command:= (Discrete_In.ManReqs3.1 OR Discrete_In.Go_Home),
			SideA_Indicator:= FALSE,
			SideB_Indicator:= FALSE,
			TurnOn_SideA_SOL=> N102.Q.0,
			TurnOn_SideB_SOL=> N102.Q.1,
			TurnOn_SideA_Indicator=> Manual_Indicators3.0,
			TurnOn_SideB_Indicator=> Manual_Indicators3.1
			 );
		Valve33FB.In_Auto_SideA_Command:= FALSE;
		Valve33FB.In_Auto_SideB_Command:= FALSE;


	(*Valve 34, A+B*)
	(*spare*)
		Valve34FB
			(
			Enable_Motion:= Enable_Motion ,
			Enable_Latch:= TRUE,					(*Enabling Runs Valve as detent type (maintained solenoids*)
			Enable_SideA_PreCharge:= FALSE,		(*Enabling Turns Side A PreCharge Active, reset when Side B is energized in Auto*)
			Enable_SideB_PreCharge:= FALSE,		(*Enabling Turns Side B PreCharge Active, reset when Side A is energized in Auto*)
			PreCharge_Time:= T#0.10S,
			Enable_Auto_Commands:= In_Auto,
			Enable_Manual_Commands:= In_Manual AND All_Robots_Clear,
			In_Manual_SideA_Command:= Discrete_In.ManReqs3.2,
			In_Manual_SideB_Command:= Discrete_In.ManReqs3.3,
			SideA_Indicator:= FALSE,
			SideB_Indicator:= FALSE,
			TurnOn_SideA_SOL=> N102.Q.2,
			TurnOn_SideB_SOL=> N102.Q.3,
			TurnOn_SideA_Indicator=> Manual_Indicators3.2,
			TurnOn_SideB_Indicator=> Manual_Indicators3.3
			 );
		Valve34FB.In_Auto_SideA_Command:= FALSE;
		Valve34FB.In_Auto_SideB_Command:= FALSE;


	(*Valve 35, A+B*)
	(*spare*)
		Valve35FB
			(
			Enable_Motion:= Enable_Motion ,
			Enable_Latch:= TRUE,					(*Enabling Runs Valve as detent type (maintained solenoids*)
			Enable_SideA_PreCharge:= FALSE,		(*Enabling Turns Side A PreCharge Active, reset when Side B is energized in Auto*)
			Enable_SideB_PreCharge:= FALSE,		(*Enabling Turns Side B PreCharge Active, reset when Side A is energized in Auto*)
			PreCharge_Time:= T#0.10S,
			Enable_Auto_Commands:= In_Auto,
			Enable_Manual_Commands:= In_Manual AND All_Robots_Clear,
			In_Manual_SideA_Command:= Discrete_In.ManReqs3.4,
			In_Manual_SideB_Command:= Discrete_In.ManReqs3.5,
			SideA_Indicator:= FALSE,
			SideB_Indicator:= FALSE,
			TurnOn_SideA_SOL=> N102.Q.4,
			TurnOn_SideB_SOL=> N102.Q.5,
			TurnOn_SideA_Indicator=> Manual_Indicators3.4,
			TurnOn_SideB_Indicator=> Manual_Indicators3.5
			 );
		Valve35FB.In_Auto_SideA_Command:= FALSE;
		Valve35FB.In_Auto_SideB_Command:= FALSE;


	(*Valve 36, A+B*)
	(*spare*)
		Valve36FB
			(
			Enable_Motion:= Enable_Motion ,
			Enable_Latch:= TRUE,					(*Enabling Runs Valve as detent type (maintained solenoids*)
			Enable_SideA_PreCharge:= FALSE,		(*Enabling Turns Side A PreCharge Active, reset when Side B is energized in Auto*)
			Enable_SideB_PreCharge:= FALSE,		(*Enabling Turns Side B PreCharge Active, reset when Side A is energized in Auto*)
			PreCharge_Time:= T#0.10S,
			Enable_Auto_Commands:= In_Auto,
			Enable_Manual_Commands:= In_Manual AND All_Robots_Clear,
			In_Manual_SideA_Command:= Discrete_In.ManReqs3.6,
			In_Manual_SideB_Command:= Discrete_In.ManReqs3.7,
			SideA_Indicator:= FALSE,
			SideB_Indicator:= FALSE,
			TurnOn_SideA_SOL=> N102.Q.6,
			TurnOn_SideB_SOL=> N102.Q.7,
			TurnOn_SideA_Indicator=> Manual_Indicators3.6,
			TurnOn_SideB_Indicator=> Manual_Indicators3.7
			 );
		Valve36FB.In_Auto_SideA_Command:= FALSE;
		Valve36FB.In_Auto_SideB_Command:= FALSE;


	(*Valve 37, A+B*)
	(*spare*)
		Valve37FB
			(
			Enable_Motion:= Enable_Motion ,
			Enable_Latch:= TRUE,					(*Enabling Runs Valve as detent type (maintained solenoids*)
			Enable_SideA_PreCharge:= FALSE,		(*Enabling Turns Side A PreCharge Active, reset when Side B is energized in Auto*)
			Enable_SideB_PreCharge:= FALSE,		(*Enabling Turns Side B PreCharge Active, reset when Side A is energized in Auto*)
			PreCharge_Time:= T#0.10S,
			Enable_Auto_Commands:= In_Auto,
			Enable_Manual_Commands:= In_Manual AND All_Robots_Clear,
			In_Manual_SideA_Command:= Discrete_In.ManReqs3.8,
			In_Manual_SideB_Command:= Discrete_In.ManReqs3.9,
			SideA_Indicator:= FALSE,
			SideB_Indicator:= FALSE,
			TurnOn_SideA_SOL=> N102.Q.8,
			TurnOn_SideB_SOL=> N102.Q.9,
			TurnOn_SideA_Indicator=> Manual_Indicators3.8,
			TurnOn_SideB_Indicator=> Manual_Indicators3.9
			 );
		Valve37FB.In_Auto_SideA_Command:= FALSE;
		Valve37FB.In_Auto_SideB_Command:= FALSE;


	(*Valve 38, A+B*)
	(*spare*)
		Valve38FB
			(
			Enable_Motion:= Enable_Motion ,
			Enable_Latch:= TRUE,					(*Enabling Runs Valve as detent type (maintained solenoids*)
			Enable_SideA_PreCharge:= FALSE,		(*Enabling Turns Side A PreCharge Active, reset when Side B is energized in Auto*)
			Enable_SideB_PreCharge:= FALSE,		(*Enabling Turns Side B PreCharge Active, reset when Side A is energized in Auto*)
			PreCharge_Time:= T#0.10S,
			Enable_Auto_Commands:= In_Auto,
			Enable_Manual_Commands:= In_Manual AND All_Robots_Clear,
			In_Manual_SideA_Command:= Discrete_In.ManReqs3.10,
			In_Manual_SideB_Command:= Discrete_In.ManReqs3.11,
			SideA_Indicator:= FALSE,
			SideB_Indicator:= FALSE,
			TurnOn_SideA_SOL=> N102.Q.10,
			TurnOn_SideB_SOL=> N102.Q.11,
			TurnOn_SideA_Indicator=> Manual_Indicators3.10,
			TurnOn_SideB_Indicator=> Manual_Indicators3.11
			 );
		Valve38FB.In_Auto_SideA_Command:= FALSE;
		Valve38FB.In_Auto_SideB_Command:= FALSE;


	(*Valve 39, A+B*)
	(*spare*)
		Valve39FB
			(
			Enable_Motion:= Enable_Motion ,
			Enable_Latch:= TRUE,					(*Enabling Runs Valve as detent type (maintained solenoids*)
			Enable_SideA_PreCharge:= FALSE,		(*Enabling Turns Side A PreCharge Active, reset when Side B is energized in Auto*)
			Enable_SideB_PreCharge:= FALSE,		(*Enabling Turns Side B PreCharge Active, reset when Side A is energized in Auto*)
			PreCharge_Time:= T#0.10S,
			Enable_Auto_Commands:= In_Auto,
			Enable_Manual_Commands:= In_Manual AND All_Robots_Clear,
			In_Manual_SideA_Command:= Discrete_In.ManReqs3.12,
			In_Manual_SideB_Command:= Discrete_In.ManReqs3.13,
			SideA_Indicator:= FALSE,
			SideB_Indicator:= FALSE,
			TurnOn_SideA_SOL=> N102.Q.12,
			TurnOn_SideB_SOL=> N102.Q.13,
			TurnOn_SideA_Indicator=> Manual_Indicators3.12,
			TurnOn_SideB_Indicator=> Manual_Indicators3.13
			 );
		Valve39FB.In_Auto_SideA_Command:= FALSE;
		Valve39FB.In_Auto_SideB_Command:= FALSE;


	(*Valve 40, A+B*)
	(*spare*)
		Valve40FB
			(
			Enable_Motion:= Enable_Motion ,
			Enable_Latch:= TRUE,					(*Enabling Runs Valve as detent type (maintained solenoids*)
			Enable_SideA_PreCharge:= FALSE,		(*Enabling Turns Side A PreCharge Active, reset when Side B is energized in Auto*)
			Enable_SideB_PreCharge:= FALSE,		(*Enabling Turns Side B PreCharge Active, reset when Side A is energized in Auto*)
			PreCharge_Time:= T#0.10S,
			Enable_Auto_Commands:= In_Auto,
			Enable_Manual_Commands:= In_Manual AND All_Robots_Clear,
			In_Manual_SideA_Command:= Discrete_In.ManReqs3.14,
			In_Manual_SideB_Command:= Discrete_In.ManReqs3.15,
			SideA_Indicator:= FALSE,
			SideB_Indicator:= FALSE,
			TurnOn_SideA_SOL=> N102.Q.14,
			TurnOn_SideB_SOL=> N102.Q.15,
			TurnOn_SideA_Indicator=> Manual_Indicators3.14,
			TurnOn_SideB_Indicator=> Manual_Indicators3.15
			 );
		Valve40FB.In_Auto_SideA_Command:= FALSE;
		Valve40FB.In_Auto_SideB_Command:= FALSE;


	(*Valve 41, A+B*)
	(*spare*)
		Valve41FB
			(
			Enable_Motion:= Enable_Motion ,
			Enable_Latch:= TRUE,					(*Enabling Runs Valve as detent type (maintained solenoids*)
			Enable_SideA_PreCharge:= FALSE,		(*Enabling Turns Side A PreCharge Active, reset when Side B is energized in Auto*)
			Enable_SideB_PreCharge:= FALSE,		(*Enabling Turns Side B PreCharge Active, reset when Side A is energized in Auto*)
			PreCharge_Time:= T#0.10S,
			Enable_Auto_Commands:= In_Auto,
			Enable_Manual_Commands:= In_Manual AND All_Robots_Clear,
			In_Manual_SideA_Command:= Discrete_In.ManReqs3.16,
			In_Manual_SideB_Command:= Discrete_In.ManReqs3.17,
			SideA_Indicator:= FALSE,
			SideB_Indicator:= FALSE,
			TurnOn_SideA_SOL=> N102.Q.16,
			TurnOn_SideB_SOL=> N102.Q.17,
			TurnOn_SideA_Indicator=> Manual_Indicators3.16,
			TurnOn_SideB_Indicator=> Manual_Indicators3.17
			 );
		Valve41FB.In_Auto_SideA_Command:= FALSE;
		Valve41FB.In_Auto_SideB_Command:= FALSE;


	(*Valve 42, A+B*)
	(*spare*)
		Valve42FB
			(
			Enable_Motion:= Enable_Motion ,
			Enable_Latch:= TRUE,					(*Enabling Runs Valve as detent type (maintained solenoids*)
			Enable_SideA_PreCharge:= FALSE,		(*Enabling Turns Side A PreCharge Active, reset when Side B is energized in Auto*)
			Enable_SideB_PreCharge:= FALSE,		(*Enabling Turns Side B PreCharge Active, reset when Side A is energized in Auto*)
			PreCharge_Time:= T#0.10S,
			Enable_Auto_Commands:= In_Auto,
			Enable_Manual_Commands:= In_Manual AND All_Robots_Clear,
			In_Manual_SideA_Command:= Discrete_In.ManReqs3.18,
			In_Manual_SideB_Command:= Discrete_In.ManReqs3.19,
			SideA_Indicator:= FALSE,
			SideB_Indicator:= FALSE,
			TurnOn_SideA_SOL=> N102.Q.18,
			TurnOn_SideB_SOL=> N102.Q.19,
			TurnOn_SideA_Indicator=> Manual_Indicators3.18,
			TurnOn_SideB_Indicator=> Manual_Indicators3.19
			 );
		Valve42FB.In_Auto_SideA_Command:= FALSE;
		Valve42FB.In_Auto_SideB_Command:= FALSE;


	(*Valve 43, A+B*)
	(*spare*)
		Valve43FB
			(
			Enable_Motion:= Enable_Motion ,
			Enable_Latch:= TRUE,					(*Enabling Runs Valve as detent type (maintained solenoids*)
			Enable_SideA_PreCharge:= FALSE,		(*Enabling Turns Side A PreCharge Active, reset when Side B is energized in Auto*)
			Enable_SideB_PreCharge:= FALSE,		(*Enabling Turns Side B PreCharge Active, reset when Side A is energized in Auto*)
			PreCharge_Time:= T#0.10S,
			Enable_Auto_Commands:= In_Auto,
			Enable_Manual_Commands:= In_Manual AND All_Robots_Clear,
			In_Manual_SideA_Command:= Discrete_In.ManReqs3.20,
			In_Manual_SideB_Command:= Discrete_In.ManReqs3.21,
			SideA_Indicator:= FALSE,
			SideB_Indicator:= FALSE,
			TurnOn_SideA_SOL=> N102.Q.20,
			TurnOn_SideB_SOL=> N102.Q.21,
			TurnOn_SideA_Indicator=> Manual_Indicators3.20,
			TurnOn_SideB_Indicator=> Manual_Indicators3.21
			 );
		Valve43FB.In_Auto_SideA_Command:= FALSE;
		Valve43FB.In_Auto_SideB_Command:= FALSE;


	(*Valve 44, A+B*)
	(*spare*)
		Valve44FB
			(
			Enable_Motion:= Enable_Motion ,
			Enable_Latch:= TRUE,					(*Enabling Runs Valve as detent type (maintained solenoids*)
			Enable_SideA_PreCharge:= FALSE,		(*Enabling Turns Side A PreCharge Active, reset when Side B is energized in Auto*)
			Enable_SideB_PreCharge:= FALSE,		(*Enabling Turns Side B PreCharge Active, reset when Side A is energized in Auto*)
			PreCharge_Time:= T#0.10S,
			Enable_Auto_Commands:= In_Auto,
			Enable_Manual_Commands:= In_Manual AND All_Robots_Clear,
			In_Manual_SideA_Command:= Discrete_In.ManReqs3.22,
			In_Manual_SideB_Command:= Discrete_In.ManReqs3.23,
			SideA_Indicator:= FALSE,
			SideB_Indicator:= FALSE,
			TurnOn_SideA_SOL=> N102.Q.22,
			TurnOn_SideB_SOL=> N102.Q.23,
			TurnOn_SideA_Indicator=> Manual_Indicators3.22,
			TurnOn_SideB_Indicator=> Manual_Indicators3.23
			 );
		Valve44FB.In_Auto_SideA_Command:= FALSE;
		Valve44FB.In_Auto_SideB_Command:= FALSE;


	(*Valve 45, A+B*)
	(*spare*)
		Valve45FB
			(
			Enable_Motion:= Enable_Motion ,
			Enable_Latch:= TRUE,					(*Enabling Runs Valve as detent type (maintained solenoids*)
			Enable_SideA_PreCharge:= FALSE,		(*Enabling Turns Side A PreCharge Active, reset when Side B is energized in Auto*)
			Enable_SideB_PreCharge:= FALSE,		(*Enabling Turns Side B PreCharge Active, reset when Side A is energized in Auto*)
			PreCharge_Time:= T#0.10S,
			Enable_Auto_Commands:= In_Auto,
			Enable_Manual_Commands:= In_Manual AND All_Robots_Clear,
			In_Manual_SideA_Command:= Discrete_In.ManReqs3.24,
			In_Manual_SideB_Command:= Discrete_In.ManReqs3.25,
			SideA_Indicator:= FALSE,
			SideB_Indicator:= FALSE,
			TurnOn_SideA_SOL=> N102.Q.24,
			TurnOn_SideB_SOL=> N102.Q.25,
			TurnOn_SideA_Indicator=> Manual_Indicators3.24,
			TurnOn_SideB_Indicator=> Manual_Indicators3.25
			 );
		Valve45FB.In_Auto_SideA_Command:= FALSE;
		Valve45FB.In_Auto_SideB_Command:= FALSE;


	(*Valve 46, A+B*)
	(*spare*)
		Valve46FB
			(
			Enable_Motion:= Enable_Motion ,
			Enable_Latch:= TRUE,					(*Enabling Runs Valve as detent type (maintained solenoids*)
			Enable_SideA_PreCharge:= FALSE,		(*Enabling Turns Side A PreCharge Active, reset when Side B is energized in Auto*)
			Enable_SideB_PreCharge:= FALSE,		(*Enabling Turns Side B PreCharge Active, reset when Side A is energized in Auto*)
			PreCharge_Time:= T#0.10S,
			Enable_Auto_Commands:= In_Auto,
			Enable_Manual_Commands:= In_Manual AND All_Robots_Clear,
			In_Manual_SideA_Command:= Discrete_In.ManReqs3.26,
			In_Manual_SideB_Command:= Discrete_In.ManReqs3.27,
			SideA_Indicator:= FALSE,
			SideB_Indicator:= FALSE,
			TurnOn_SideA_SOL=> N102.Q.26,
			TurnOn_SideB_SOL=> N102.Q.27,
			TurnOn_SideA_Indicator=> Manual_Indicators3.26,
			TurnOn_SideB_Indicator=> Manual_Indicators3.27
			 );
		Valve46FB.In_Auto_SideA_Command:= FALSE;
		Valve46FB.In_Auto_SideB_Command:= FALSE;


	(*Valve 47, A+B*)
	(*spare*)
		Valve47FB
			(
			Enable_Motion:= Enable_Motion ,
			Enable_Latch:= TRUE,					(*Enabling Runs Valve as detent type (maintained solenoids*)
			Enable_SideA_PreCharge:= FALSE,		(*Enabling Turns Side A PreCharge Active, reset when Side B is energized in Auto*)
			Enable_SideB_PreCharge:= FALSE,		(*Enabling Turns Side B PreCharge Active, reset when Side A is energized in Auto*)
			PreCharge_Time:= T#0.10S,
			Enable_Auto_Commands:= In_Auto,
			Enable_Manual_Commands:= In_Manual AND All_Robots_Clear,
			In_Manual_SideA_Command:= Discrete_In.ManReqs3.28,
			In_Manual_SideB_Command:= Discrete_In.ManReqs3.29,
			SideA_Indicator:= FALSE,
			SideB_Indicator:= FALSE,
			TurnOn_SideA_SOL=> N102.Q.28,
			TurnOn_SideB_SOL=> N102.Q.29,
			TurnOn_SideA_Indicator=> Manual_Indicators3.28,
			TurnOn_SideB_Indicator=> Manual_Indicators3.29
			 );
		Valve47FB.In_Auto_SideA_Command:= FALSE;
		Valve47FB.In_Auto_SideB_Command:= FALSE;


	(*Valve 48, A+B*)
	(*spare*)
		Valve48FB
			(
			Enable_Motion:= Enable_Motion ,
			Enable_Latch:= TRUE,					(*Enabling Runs Valve as detent type (maintained solenoids*)
			Enable_SideA_PreCharge:= FALSE,		(*Enabling Turns Side A PreCharge Active, reset when Side B is energized in Auto*)
			Enable_SideB_PreCharge:= FALSE,		(*Enabling Turns Side B PreCharge Active, reset when Side A is energized in Auto*)
			PreCharge_Time:= T#0.10S,
			Enable_Auto_Commands:= In_Auto,
			Enable_Manual_Commands:= In_Manual AND All_Robots_Clear,
			In_Manual_SideA_Command:= Discrete_In.ManReqs3.30,
			In_Manual_SideB_Command:= Discrete_In.ManReqs3.31,
			SideA_Indicator:= FALSE,
			SideB_Indicator:= FALSE,
			TurnOn_SideA_SOL=> N102.Q.30,
			TurnOn_SideB_SOL=> N102.Q.31,
			TurnOn_SideA_Indicator=> Manual_Indicators3.30,
			TurnOn_SideB_Indicator=> Manual_Indicators3.31
			 );
		Valve48FB.In_Auto_SideA_Command:= FALSE;
		Valve48FB.In_Auto_SideB_Command:= FALSE;


























(*end*)
END_ACTION

ACTION Xfer_To_UI:
(*Transfer General Status of Fixture and I/O Images for Display On HMI*)
	Discrete_Image.Status:= Status;
	Discrete_Image.CLFaults1:= CLFaults1;
	Discrete_Image.CLFaults2:= CLFaults2;
	Discrete_Image.CLFaults3:= CLFaults3;
	Discrete_Image.CLFaults4:= CLFaults4;
	Discrete_Image.CLFaulted:= CLFaulted;
	Discrete_Image.PPFaults:= PPFaults;
	Discrete_Image.PPFaults1:= PPFaults1;
	Discrete_Image.PPFaults2:= PPFaults2;
	Discrete_Image.PPFaulted:= PPFaulted;
	Discrete_Image.Model_Data:= Model_ID;
	Discrete_Image.ToolID:= Fix_ID;
	Discrete_Image.ProdCount:= Prod_Count_Out;
	Discrete_Image.CycleTime:= Cycle_Time_Out;
	Discrete_Image.PrevCycleTime:= PrevCycle_Time_Out;
	Discrete_Image.LoadTime:= Load_Time_Out;
	Discrete_Image.WeldTime:= Weld_Time_Out;
	Discrete_Image.UnloadTime:= Unload_Time_Out;

	Discrete_Image.InAuto:= In_Auto_Mode;
	Discrete_Image.InManual:= In_Manual_Mode;
	Discrete_Image.ManInds:= Manual_Indicators1;
	Discrete_Image.ManInds2:= Manual_Indicators2;
	Discrete_Image.ManInds3:= Manual_Indicators3;
	Discrete_Image.At_Home:= Tool_At_Home;
	Discrete_Image.Enable_Motion:= Enable_Motion;
	Discrete_Image.All_Sensors_Off:= All_Sensors_Off;
	Discrete_Image.Bypass_ACKS:= Discrete_In.Bypass_REQS;
	Discrete_Image.CustomApplication_ACKS:= Discrete_In.CustomApplication_REQS;
	Discrete_Image.Fixture_Allow_Model_Change:= Fixture_Allow_Model_Change;
	Discrete_Image.NodeLayout:=NodeLayout;
	Discrete_Image.NodeState:=NodeState;
	
	Discrete_Image.Input_Node_Count:= Discrete_In.Input_Node_Count;
	Discrete_Image.VB_Node_Count:= Discrete_In.VB_Node_Count;
	Discrete_Image.Water_Stand_Count:= Discrete_In.Water_Stand_Count;

	IF  (Discrete_Image.Input_Node_Count < 4)
		THEN Discrete_Image.VB_Screen_Position:= 1;
	ELSIF  (Discrete_Image.Input_Node_Count < 7)
		THEN Discrete_Image.VB_Screen_Position:= 2;
	ELSIF  (Discrete_Image.Input_Node_Count < 10)
		THEN Discrete_Image.VB_Screen_Position:= 3;
	ELSIF  (Discrete_Image.Input_Node_Count < 13)
		THEN Discrete_Image.VB_Screen_Position:= 4;
	ELSIF  (Discrete_Image.Input_Node_Count < 16)
		THEN Discrete_Image.VB_Screen_Position:= 5;
	ELSIF  (Discrete_Image.Input_Node_Count < 19)
		THEN Discrete_Image.VB_Screen_Position:= 6;
	ELSIF  (Discrete_Image.Input_Node_Count < 22)
		THEN Discrete_Image.VB_Screen_Position:= 7;
	ELSIF  (Discrete_Image.Input_Node_Count < 26)
		THEN Discrete_Image.VB_Screen_Position:= 8;
	ELSE
			Discrete_Image.VB_Screen_Position:= 9;
	END_IF;

	Discrete_Image.N00:= N00;
	Discrete_Image.N01:= N01;
	Discrete_Image.N02:= N02;
	Discrete_Image.N03:= N03;
	Discrete_Image.N04:= N04;
	Discrete_Image.N05:= N05;
	Discrete_Image.N06:= N06;
	Discrete_Image.N07:= N07;
	Discrete_Image.N08:= N08;
	Discrete_Image.N09:= N09;
	Discrete_Image.N10:= N10;
	Discrete_Image.N11:= N11;
	Discrete_Image.N12:= N12;
	Discrete_Image.N13:= N13;
	Discrete_Image.N14:= N14;
	Discrete_Image.N15:= N15;
	Discrete_Image.N16:= N16;
	Discrete_Image.N17:= N17;
	Discrete_Image.N18:= N18;
	Discrete_Image.N19:= N19;
	Discrete_Image.N100:= N100;
	Discrete_Image.N100_STAT:= N100_STAT;
	Discrete_Image.N101:= N101;
	Discrete_Image.N101_STAT:= N101_STAT;
	Discrete_Image.N102:= N102;
	Discrete_Image.N102_STAT:= N102_STAT;


	Discrete_Image.ECatSlave_Cable_Breaks:= ECatSlave_Cable_Breaks;

	Discrete_Image.Operator_Performance_Pen:= Production_Report.Shift_Report[0].Prod_Performance;
END_ACTION

END_PROGRAM

// ---- POUs/Fixtures and EOAT/Not_Used/Fix13.TcPOU
(*Fixture*)

PROGRAM Fix13
	VAR_INPUT
		Enable_Prog: BOOL;
		Enable_Motion: BOOL;
		Discrete_In: udt_FixXX_Input_Image_20180202;
		Dry_Cycle: BOOL;
		Cell_In_Services: BOOL;
		Flash_Rate: BOOL;
		NodeLayout:udt_ECATNodeData_20221507;

	END_VAR

	VAR
(*Hardware Related Data Types*)
			(*Develop "Beckhoff Nodes"*)
			{attribute 'OPC.UA.DA':='1'}
			N00 AT %I*: udt_EP1111;
			{attribute 'OPC.UA.DA':='1'}
			N01 AT %I*: udt_EP1008_002_v2;
			{attribute 'OPC.UA.DA':='1'}
			N02 AT %I*: udt_EP1008_002_v2;
			{attribute 'OPC.UA.DA':='1'}
			N03 AT %I*: udt_EP1008_002_v2;
			{attribute 'OPC.UA.DA':='1'}
			N04 AT %I*: udt_EP1008_002_v2;
			{attribute 'OPC.UA.DA':='1'}
			N05 AT %I*: udt_EP1008_002_v2;
			{attribute 'OPC.UA.DA':='1'}
			N06 AT %I*: udt_EP1008_002_v2;
			{attribute 'OPC.UA.DA':='1'}
			N07 AT %I*: udt_EP1008_002_v2;
			{attribute 'OPC.UA.DA':='1'}
			N08 AT %I*: udt_EP1008_002_v2;
			{attribute 'OPC.UA.DA':='1'}
			N09 AT %I*: udt_EP1008_002_v2;
			{attribute 'OPC.UA.DA':='1'}
			N10 AT %I*: udt_EP1008_002_v2;
			{attribute 'OPC.UA.DA':='1'}
			N11 AT %I*: udt_EP1008_002_v2;
			{attribute 'OPC.UA.DA':='1'}
			N12 AT %I*: udt_EP1008_002_v2;
			{attribute 'OPC.UA.DA':='1'}
			N13 AT %I*: udt_EP1008_002_v2;
			{attribute 'OPC.UA.DA':='1'}
			N14 AT %I*: udt_EP1008_002_v2;
			{attribute 'OPC.UA.DA':='1'}
			N15 AT %I*: udt_EP1008_002_v2;
			{attribute 'OPC.UA.DA':='1'}
			N16 AT %I*: udt_EP1008_002_v2;
			{attribute 'OPC.UA.DA':='1'}
			N17 AT %I*: udt_EP1008_002_v2;
			{attribute 'OPC.UA.DA':='1'}
			N18 AT %I*: udt_EP1008_002_v2;
			{attribute 'OPC.UA.DA':='1'}
			N19 AT %I*: udt_EP1008_002_v2;
			{attribute 'OPC.UA.DA':='1'}
			N20 AT %I*: udt_EP1008_002_v2;
			{attribute 'OPC.UA.DA':='1'}
			N21 AT %I*: udt_EP1008_002_v2;
			{attribute 'OPC.UA.DA':='1'}
			N22 AT %I*: udt_EP1008_002_v2;
			{attribute 'OPC.UA.DA':='1'}
			N100 AT %Q*: udt_SMC_EX260_ValveBank;
			{attribute 'OPC.UA.DA':='1'}
			N100_STAT AT %I*:udt_SMC_EX260_Stat;
			{attribute 'OPC.UA.DA':='1'}
			N101 AT %Q*: udt_SMC_EX260_ValveBank;
			{attribute 'OPC.UA.DA':='1'}
			N101_STAT AT %I*:udt_SMC_EX260_Stat;
			{attribute 'OPC.UA.DA':='1'}
			N102 AT %Q*: udt_SMC_EX260_ValveBank;
			{attribute 'OPC.UA.DA':='1'}
			N102_STAT AT %I*:udt_SMC_EX260_Stat;

(* Nodes States*)
		NodeState: ARRAY[0..63] OF UINT;
		DiscreteNode_OK: BOOL;
(*Cable Break States*)
		ECatSlave_Cable_Breaks: ARRAY[0..1] OF DINT;
(*Standard Internal Variables*)
		(*Generic Sensor Variables*)
		All_Sensors_On: UINT;
		All_Sensors_Off: BOOL;
		All_Sensors_Off1: BOOL;
		All_Sensors_Off2: BOOL;
		(*Generic Position Variables*)
		Tool_At_Home: BOOL;
		Tool_At_Load: UINT;
		Tool_At_Weld: UINT;
		Tool_At_Rotate: UINT;
		Tool_At_Seal: UINT;
		Tool_At_Stud: UINT;
		Tool_At_Unload: UINT ;
		(*Grouping Of Items*)
		All_QAChecks_OK: BOOL;
		QAChecks_Failed: BOOL;
		(*General Internals*)
		In_Auto: BOOL;
		In_Manual: BOOL;

		Auto_Run: BOOL;
		Reset_All_Completes:BOOL;
		Load_Robots_Clear1: BOOL;
		Load_Robots_Clear2: BOOL;
		Load_Robots_Clear: BOOL;
		Load_Robots_WorkingOK1: BOOL;
		Load_Robots_WorkingOK2: BOOL;
		Load_Robots_Complete1: BOOL;
		Load_Robots_Complete2: BOOL;
		Load_Robots_PartInEOAT1: BOOL;
		Load_Robots_PartInEOAT2: BOOL;
		Load_Robots_UnclampEarly1: BOOL;
		Load_Robots_UnclampEarly2: BOOL;
		Seal_Robots_Clear: BOOL;
		Seal_Robots_WorkingOK: BOOL;
		Seal_Robots_UnclampEarly: BOOL;
		Seal_Robots_Complete: BOOL;
		Stud_Robots_Clear: BOOL;
		Stud_Robots_WorkingOK: BOOL;
		Stud_Robots_UnclampEarly: BOOL;
		Stud_Robots_Complete: BOOL;
		Weld_Robots_Clear: BOOL;
		Weld_Robots_WorkingOK: BOOL;
		Weld_Robots_UnclampEarly: BOOL;
		Weld_Robots_Complete: BOOL;
		Mig_Robots_Ready :BOOL;
		TurntableA_Clear: BOOL;
		TurntableB_Clear: BOOL;
		Turntable_Clear:BOOL;
		Turntable_WorkingOK: BOOL;
		TurntableA_Complete: BOOL;
		TurntableB_Complete: BOOL;
		Unload_Robots_Clear1: BOOL;
		Unload_Robots_WorkingOK1: BOOL;
		Unload_Robots_Complete1: BOOL;
		Unload_Robots_EOATEmpty1: BOOL;
		Unload_Robots_Clear2: BOOL;
		Unload_Robots_WorkingOK2: BOOL;
		Unload_Robots_Complete2: BOOL;
		Unload_Robots_EOATEmpty2: BOOL;
		Unload_Robots_Clear: BOOL;
		All_Robots_Clear: BOOL;

		Unload_Robot_Complete: BOOL;

		Start_Load_Robots1: BOOL;
		Start_Load_Robots2: BOOL;
		Start_Weld_Robots: BOOL;
		Start_Unload_Robots1: BOOL;
		Start_Unload_Robots2: BOOL;
		Start_Seal_Robots: BOOL;
		Start_Stud_Robots: BOOL;
		Start_TurntableA: BOOL;
		Start_TurntableB: BOOL;
		Load_Robots_Proceed1: BOOL;
		Load_Robots_Proceed2: BOOL;
		Weld_Robots_Proceed: BOOL;
		Seal_Robots_Proceed: BOOL;
		Stud_Robots_Proceed: BOOL;
		Unload_Robots_Proceed1: BOOL;
		Unload_Robots_Proceed2: BOOL;

		Prod_Inc: R_TRIG;
		Cycle_Time: TON;
		Cycle_Time_Pulse: R_TRIG;
		Load_Time: TON;
		Weld_Time: TON;
		Seal_Time: TON;
		Stud_Time: TON;
		Turn_Time: TON;
		Unload_Time: TON;
		Date_Stamp_TMR: TON;
		Date_StampHome_TMR: TON;
		CLFaulted: UDINT;
		PPFaulted: UDINT;
		Manual_Ind_HomePrompt: BOOL;
		Fixture_Allow_Model_Change: BOOL;

(*Non-Standard Variables*)

		(*FB Instances*)
		Clamp1FB: FB_Cylinder_Status;
		Clamp2FB: FB_Cylinder_Status;
		Clamp3FB: FB_Cylinder_Status;
		Clamp4FB: FB_Cylinder_Status;
		Clamp5FB: FB_Cylinder_Status;
		Clamp6FB: FB_Cylinder_Status;
		Clamp7FB: FB_Cylinder_Status;
		Clamp8FB: FB_Cylinder_Status;
		Clamp9FB: FB_Cylinder_Status;
		Clamp10FB: FB_Cylinder_Status;
		Clamp11FB: FB_Cylinder_Status;
		Clamp12FB: FB_Cylinder_Status;
		Clamp13FB: FB_Cylinder_Status;
		Clamp14FB: FB_Cylinder_Status;
		Clamp15FB: FB_Cylinder_Status;
		Clamp16FB: FB_Cylinder_Status;
		Clamp17FB: FB_Cylinder_Status;
		Clamp18FB: FB_Cylinder_Status;
		Clamp19FB: FB_Cylinder_Status;
		Clamp20FB: FB_Cylinder_Status;
		Clamp21FB: FB_Cylinder_Status;
		Clamp22FB: FB_Cylinder_Status;
		Clamp23FB: FB_Cylinder_Status;
		Clamp24FB: FB_Cylinder_Status;
		Cyl1FB: FB_TripleCylinder_20150625;
		Pin1FB: FB_Cylinder_Status;
		Pin2FB: FB_Cylinder_Status;
		Pin3FB: FB_Cylinder_Status;
		Pin4FB: FB_Cylinder_Status;
		Pin5FB: FB_Cylinder_Status;
		Pin6FB: FB_Cylinder_Status;
		Pin7FB: FB_Cylinder_Status;
		Pin8FB: FB_Cylinder_Status;
		Pin9FB: FB_Cylinder_Status;
		Pin10FB: FB_Cylinder_Status;
		Pin11FB: FB_Cylinder_Status;
		Pin12FB: FB_Cylinder_Status;
		Pin13FB: FB_Cylinder_Status;
		Pin14FB: FB_Cylinder_Status;
		Slide1FB: FB_Cylinder_Status;
		Slide2FB: FB_Cylinder_Status;
		Slide3FB: FB_Cylinder_Status;
		Slide4FB: FB_Cylinder_Status;
		Slide5FB: FB_Cylinder_Status;
		Slide6FB: FB_Cylinder_Status;
		Swing1FB: FB_Cylinder_Status;
		Swing2FB: FB_Cylinder_Status;
		Swing3FB: FB_Cylinder_Status;
		Swing4FB: FB_Cylinder_Status;
		Swing5FB: FB_Cylinder_Status;
		Swing6FB: FB_Cylinder_Status;
		QACheck1FB: FB_Cylinder_Status;
		QACheck2FB: FB_Cylinder_Status;
		CheckQA1FB: FB_GTAC_QAcheck_20150529;
		Part_Present1FB: FB_PP_Sensor;
		Part_Present2FB: FB_PP_Sensor;
		Part_Present3FB: FB_PP_Sensor;
		Part_Present4FB: FB_PP_Sensor;
		Part_Present5FB: FB_PP_Sensor;
		Part_Present6FB: FB_PP_Sensor;
		Part_Present7FB: FB_PP_Sensor;
		Part_Present8FB: FB_PP_Sensor;
		Part_Present9FB: FB_PP_Sensor;
		Part_Present10FB: FB_PP_Sensor;
		Part_Present11FB: FB_PP_Sensor;
		Part_Present12FB: FB_PP_Sensor;
		Part_Present13FB: FB_PP_Sensor;
		Part_Present14FB: FB_PP_Sensor;
		Part_Present15FB: FB_PP_Sensor;
		Part_Present16FB: FB_PP_Sensor;
		Part_Present17FB: FB_PP_Sensor;
		Part_Present18FB: FB_PP_Sensor;
		Part_Present19FB: FB_PP_Sensor;
		Part_Present20FB: FB_PP_Sensor;
		Part_Present21FB: FB_PP_Sensor;
		Part_Present22FB: FB_PP_Sensor;
		Part_Present23FB: FB_PP_Sensor;
		Part_Present24FB: FB_PP_Sensor;
		Part_Present25FB: FB_PP_Sensor;
		Part_Present26FB: FB_PP_Sensor;
		Part_Present27FB: FB_PP_Sensor;
		Part_Present28FB: FB_PP_Sensor;
		Part_Present29FB: FB_PP_Sensor;
		Part_Present30FB: FB_PP_Sensor;
		Part_Present31FB: FB_PP_Sensor;
		Part_Present32FB: FB_PP_Sensor;
		Part_Present33FB: FB_PP_Sensor;
		Part_Present34FB: FB_PP_Sensor;
		Part_Present35FB: FB_PP_Sensor;
		Part_Present36FB: FB_PP_Sensor;
		Part_Present37FB: FB_PP_Sensor;
		Part_Present38FB: FB_PP_Sensor;
		Part_Present39FB: FB_PP_Sensor;
		Part_Present40FB: FB_PP_Sensor;
		Tape_Present1FB: FB_PP_Sensor;

		(*Valve FBs*)
		Valve1FB: FB_GTAC_Valve_20170704;
		Valve2FB: FB_GTAC_Valve_20170704;
		Valve3FB: FB_GTAC_Valve_20170704;
		Valve4FB: FB_GTAC_Valve_20170704;
		Valve5FB: FB_GTAC_Valve_20170704;
		Valve6FB: FB_GTAC_Valve_20170704;
		Valve7FB: FB_GTAC_Valve_20170704;
		Valve8FB: FB_GTAC_Valve_20170704;
		Valve9FB: FB_GTAC_Valve_20170704;
		Valve10FB: FB_GTAC_Valve_20170704;
		Valve11FB: FB_GTAC_Valve_20170704;
		Valve12FB: FB_GTAC_Valve_20170704;
		Valve13FB: FB_GTAC_Valve_20170704;
		Valve14FB: FB_GTAC_Valve_20170704;
		Valve15FB: FB_GTAC_Valve_20170704;
		Valve16FB: FB_GTAC_Valve_20170704;
		Valve17FB: FB_GTAC_Valve_20170704;
		Valve18FB: FB_GTAC_Valve_20170704;
		Valve19FB: FB_GTAC_Valve_20170704;
		Valve20FB: FB_GTAC_Valve_20170704;
		Valve21FB: FB_GTAC_Valve_20170704;
		Valve22FB: FB_GTAC_Valve_20170704;
		Valve23FB: FB_GTAC_Valve_20170704;
		Valve24FB: FB_GTAC_Valve_20170704;
		Valve25FB: FB_GTAC_Valve_20170704;
		Valve26FB: FB_GTAC_Valve_20170704;
		Valve27FB: FB_GTAC_Valve_20170704;
		Valve28FB: FB_GTAC_Valve_20170704;
		Valve29FB: FB_GTAC_Valve_20170704;
		Valve30FB: FB_GTAC_Valve_20170704;
		Valve31FB: FB_GTAC_Valve_20170704;
		Valve32FB: FB_GTAC_Valve_20170704;
		Valve33FB: FB_GTAC_Valve_20170704;
		Valve34FB: FB_GTAC_Valve_20170704;
		Valve35FB: FB_GTAC_Valve_20170704;
		Valve36FB: FB_GTAC_Valve_20170704;
		Valve37FB: FB_GTAC_Valve_20170704;
		Valve38FB: FB_GTAC_Valve_20170704;
		Valve39FB: FB_GTAC_Valve_20170704;
		Valve40FB: FB_GTAC_Valve_20170704;
		Valve41FB: FB_GTAC_Valve_20170704;
		Valve42FB: FB_GTAC_Valve_20170704;
		Valve43FB: FB_GTAC_Valve_20170704;
		Valve44FB: FB_GTAC_Valve_20170704;
		Valve45FB: FB_GTAC_Valve_20170704;
		Valve46FB: FB_GTAC_Valve_20170704;
		Valve47FB: FB_GTAC_Valve_20170704;
		Valve48FB: FB_GTAC_Valve_20170704;

		(*Tool Positions*)
			(*Add User Indivdual Position Variables Here*)
			Clamp1ADVD: BOOL;
			Clamp1RETD: BOOL;
			Clamp2ADVD: BOOL;
			Clamp2RETD: BOOL;
			Clamp3ADVD: BOOL;
			Clamp3RETD: BOOL;
			Clamp4ADVD: BOOL;
			Clamp4RETD: BOOL;
			Clamp5ADVD: BOOL;
			Clamp5RETD: BOOL;
			Clamp6ADVD: BOOL;
			Clamp6RETD: BOOL;
			Clamp7ADVD: BOOL;
			Clamp7RETD: BOOL;
			Clamp8ADVD: BOOL;
			Clamp8RETD: BOOL;
			Clamp9ADVD: BOOL;
			Clamp9RETD: BOOL;
			Clamp10ADVD: BOOL;
			Clamp10RETD: BOOL;
			Clamp11ADVD: BOOL;
			Clamp11RETD: BOOL;
			Clamp12ADVD: BOOL;
			Clamp12RETD: BOOL;
			Clamp13ADVD: BOOL;
			Clamp13RETD: BOOL;
			Clamp14ADVD: BOOL;
			Clamp14RETD: BOOL;
			Clamp15ADVD: BOOL;
			Clamp15RETD: BOOL;
			Clamp16ADVD: BOOL;
			Clamp16RETD: BOOL;
			Clamp17ADVD: BOOL;
			Clamp17RETD: BOOL;
			Clamp18ADVD: BOOL;
			Clamp18RETD: BOOL;
			Clamp19ADVD: BOOL;
			Clamp19RETD: BOOL;
			Clamp20ADVD: BOOL;
			Clamp20RETD: BOOL;
			Clamp21ADVD: BOOL;
			Clamp21RETD: BOOL;
			Clamp22ADVD: BOOL;
			Clamp22RETD: BOOL;
			Clamp23ADVD: BOOL;
			Clamp23RETD: BOOL;
			Clamp24ADVD: BOOL;
			Clamp24RETD: BOOL;
			Cyl1ADVD: BOOL;
			Cyl1MID: BOOL;
			Cyl1RETD: BOOL;
			Pin1ADVD: BOOL;
			Pin1RETD: BOOL;
			Pin2ADVD: BOOL;
			Pin2RETD: BOOL;
			Pin3ADVD: BOOL;
			Pin3RETD: BOOL;
			Pin4ADVD: BOOL;
			Pin4RETD: BOOL;
			Pin5ADVD: BOOL;
			Pin5RETD: BOOL;
			Pin6ADVD: BOOL;
			Pin6RETD: BOOL;
			Pin7ADVD: BOOL;
			Pin7RETD: BOOL;
			Pin8ADVD: BOOL;
			Pin8RETD: BOOL;
			Pin9ADVD: BOOL;
			Pin9RETD: BOOL;
			Pin10ADVD: BOOL;
			Pin10RETD: BOOL;
			Pin11ADVD: BOOL;
			Pin11RETD: BOOL;
			Pin12ADVD: BOOL;
			Pin12RETD: BOOL;
			Pin13ADVD: BOOL;
			Pin13RETD: BOOL;
			Pin14ADVD: BOOL;
			Pin14RETD: BOOL;
			Slide1ADVD: BOOL;
			Slide1RETD: BOOL;
			Slide2ADVD: BOOL;
			Slide2RETD: BOOL;
			Slide3ADVD: BOOL;
			Slide3RETD: BOOL;
			Slide4ADVD: BOOL;
			Slide4RETD: BOOL;
			Slide5ADVD: BOOL;
			Slide5RETD: BOOL;
			Slide6ADVD: BOOL;
			Slide6RETD: BOOL;
			Swing1ADVD: BOOL;
			Swing1RETD: BOOL;
			Swing2ADVD: BOOL;
			Swing2RETD: BOOL;
			Swing3ADVD: BOOL;
			Swing3RETD: BOOL;
			Swing4ADVD: BOOL;
			Swing4RETD: BOOL;
			Swing5ADVD: BOOL;
			Swing5RETD: BOOL;
			Swing6ADVD: BOOL;
			Swing6RETD: BOOL;
			QACheck1ADVD: BOOL;
			QACheck1RETD: BOOL;
			QACheck2ADVD: BOOL;
			QACheck2RETD: BOOL;

		(*Part Present Sensors*)
			(*Main Body Present*)
			Part_Present1: BOOL;
			Part_Present2: BOOL;
			Part_Present3: BOOL;
			Part_Present4: BOOL;
			Part_Present5: BOOL;
			Part_Present6: BOOL;
			Part_Present7: BOOL;
			Part_Present8: BOOL;
			Part_Present9: BOOL;
			Part_Present10: BOOL;
			Part_Present11: BOOL;
			Part_Present12: BOOL;
			Part_Present13: BOOL;
			Part_Present14: BOOL;
			Part_Present15: BOOL;
			Part_Present16: BOOL;
			Part_Present17: BOOL;
			Part_Present18: BOOL;
			Part_Present19: BOOL;
			Part_Present20: BOOL;
			Part_Present21: BOOL;
			Part_Present22: BOOL;
			Part_Present23: BOOL;
			Part_Present24: BOOL;
			Part_Present25: BOOL;
			Part_Present26: BOOL;
			Part_Present27: BOOL;
			Part_Present28: BOOL;
			Part_Present29: BOOL;
			Part_Present30: BOOL;
			Part_Present31: BOOL;
			Part_Present32: BOOL;
			Part_Present33: BOOL;
			Part_Present34: BOOL;
			Part_Present35: BOOL;
			Part_Present36: BOOL;
			Part_Present37: BOOL;
			Part_Present38: BOOL;
			Part_Present39: BOOL;
			Part_Present40: BOOL;
			Tape_Present1: BOOL;

		(*Motion Sequence Variables*)
			Clamp_Step: UINT;
			Repo1_Step: UINT;
			Repo2_Step: UINT;
			Repo3_Step: UINT;
			Repo4_Step: UINT;
			Unclamp_Step: UINT;

		(*Custom Application Variables*)
			Weld_Curtain_Bypass: BOOL;
			Vacuum_Bypass: BOOL;
			Sealer_Bypass: BOOL;
			Stud_Bypass: BOOL;
			Turntable_Bypassed: BOOL;
			Door_Open: BOOL;

END_VAR

	(*data that needs to be retained in the event of a power cycle*)
	VAR PERSISTENT

		Load_Complete1: BOOL;
		Load_Complete2: BOOL;
		Load_Complete: BOOL;
		Stud_Complete: BOOL;
		Welding_Complete: BOOL;
		Sealing_Complete: BOOL;
		Unload_Complete: BOOL;
		TurnA_Complete: BOOL;
		TurnB_Complete: BOOL;
		Cycle_Complete: BOOL;
		Eject_Complete: BOOL;
		VacCheck_Complete: BOOL;
		Date_Stamp_Complete: BOOL;
		Load_Seq01: FB_GTAC_Load_Seq_20230302;
		Production_Count:INT;
		Repo_REQS: UINT;
		(*Allow_Load_PreCall: BOOL;
		Allow_Weld_PreCall: BOOL;
		Allow_Unload_PreCall: BOOL;*)
		(*All_SubPP_Off: BOOL;*)
		Production_Report: FB_Production_Report_20221007;

	END_VAR

	VAR_OUTPUT

		Prog_Ok: BOOL;
		Discrete_Image: udt_FixXX_Output_Image_20220715;
		In_Auto_Mode: BOOL;
		In_Manual_Mode: BOOL;
		Manual_Indicators1: DINT;
		Manual_Indicators2: DINT;
		Manual_Indicators3: DINT;
		At_Home: BOOL;
		Ready_To_Load: BOOL;
		Red_Lamp_Req: BOOL;
		Status: UINT;
		CLFaults1:UDINT;
		CLFaults2:UDINT;
		CLFaults3:UDINT;
		CLFaults4:UDINT;
		PPFaults: UDINT;
		PPFaults1: UDINT;
		PPFaults2: UDINT;
		Prod_Count_Out: INT;
		Cycle_Time_Out: TIME;
		PrevCycle_Time_Out: TIME;
		Load_Time_Out: TIME;
		Weld_Time_Out: TIME;
		Seal_Time_Out: TIME;
		Stud_Time_Out: TIME;
		Turn_Time_Out: TIME;
		Unload_Time_Out: TIME;
		Model_ID: UINT;
		TurntableA_At_Robot: BOOL;
		TurntableB_At_Robot: BOOL;
		Tool_Call_ForLoadRobots1: BOOL;
		Tool_Call_ForLoadRobots2: BOOL;
		Tool_Call_ForSealRobots: BOOL;
		Tool_Call_ForStudRobots: BOOL;
		Tool_Call_ForWeldRobots: BOOL;
		Tool_Call_ForSweepA: BOOL;
		Tool_Call_ForSweepB: BOOL;
		Tool_Call_ForUnloadRobots1: BOOL;
		Tool_Call_ForUnloadRobots2: BOOL;
		Robots_Clear_ToProceed: BOOL;
		Task_ID: UINT;
		Fix_ID: UINT;
		Load_Complete1_Ack: BOOL;
		Load_Complete2_Ack: BOOL;
		Seal_Complete_Ack: BOOL;
		Stud_Complete_Ack: BOOL;
		Weld_Complete_Ack: BOOL;
		TurnA_Complete_Ack: BOOL;
		TurnB_Complete_Ack: BOOL;
		Unload_Complete1_Ack: BOOL;
		Unload_Complete2_Ack: BOOL;
		Repo_Ack: UINT;
		Door_Close_Req: BOOL;
		Door_Open_Req: BOOL;
	END_VAR

	(*Set FB_OK to True*)
	Prog_OK:= TRUE;


	(*Set conditions to allow model change*)
	Fixture_Allow_Model_Change:= (In_Manual AND Tool_At_Home AND All_Sensors_Off AND All_Robots_Clear)
							OR (Model_ID=0);



(*$$$$$$$$$$$$$$$$$$$$$$$$$$$$$$$$$$$$$$$$$$$$ Fixture Bypasses $$$$$$$$$$$$$$$$$$$$$$$$$$$$$$$$$$$$$$$$$$$$$$$$$$$$*)
	Weld_Curtain_Bypass:= Discrete_In.Bypass_REQS.0;
	Vacuum_Bypass:= Discrete_In.Bypass_REQS.1;
	Stud_Bypass:= Discrete_In.Bypass_REQS.2;
	Turntable_Bypassed:= ((TurntableA_At_Robot AND Tool_At_Home AND All_Sensors_OFF)
					OR (Turntable_Bypassed AND NOT TurntableB_At_Robot))
					OR Discrete_In.Bypass_REQS.3;
	Sealer_Bypass:= MAIN.SL01.Disp1_Bypass;


(*$$$$$$$$$$$$$$$$$$$$$$$$$$$$$$$$$$$$$$$$$$$$ Gather Status Of Hardware $$$$$$$$$$$$$$$$$$$$$$$$$$$$$$$$$$$$$$$$$$$$$$$$$$$$*)
	(*Check on Status of Hardware*)
	Hardware();

(*$$$$$$$$$$$$$$$$$$$$$$$$$$$$$$$$$$$$$$$$$$$$$ Gather Standard Inputs $$$$$$$$$$$$$$$$$$$$$$$$$$$$$$$$$$$$$$$$$$$$$$$$$$$$$$$$$*)

(*Clamp/Cylinder Inputs*)
	Cylinders();

(*Part Present Inputs*)
	Proxies();

(*$$$$$$$$$$$$$$$$$$$$$$$$$$$$$$$$$$$$$$$$$$$ Qaulity Checking Routines $$$$$$$$$$$$$$$$$$$$$$$$$$$$$$$$$$$$$$$$$$$$$$$$$$$$$$$$$*)

	(*QA Checks*)
		CheckQA1FB(
			Start_QAcheck:= Auto_Run AND Enable_Motion AND Tool_At_Load.3,
			QAcheck_Reset:= Cycle_Complete OR (In_Manual AND Discrete_In.Go_Home AND All_Sensors_Off),
			QAcheck_Retry:= In_From_ICxx.QA_Reset.0,
			QAcheck_Release:= In_From_ICxx.QA_Reset.1,
			QAcheck_Adv_In:= QACheck1ADVD AND QACheck2ADVD,
			QAcheck_Ret_In:= QACheck1RETD AND QACheck2RETD,
			User_Dry_Cycle:= Dry_Cycle,
			QAcheck_OK_Delay:= T#0.75s,
			QAcheck_Fault_Delay:= T#3.0s,
			QAcheck_OK=> All_QAChecks_OK,
			QAcheck_Failed=> QAChecks_Failed);



(*$$$$$$$$$$$$$$$$$$$$$$$$$$$$$$$$$$$$$$$$$$$$$$$$ Internal Code $$$$$$$$$$$$$$$$$$$$$$$$$$$$$$$$$$$$$$$$$$$$$$$$$$$$$$$$$$$$$$$$$$$$*)
(*Auto / Manual Mode Code*)
	IF Discrete_In.Mode_Select.0 AND NOT Discrete_In.Mode_Select.1
		THEN
			In_Auto:= TRUE;
			In_Auto_Mode:= TRUE;
	END_IF;
	IF NOT Discrete_In.Mode_Select.0 AND Discrete_In.Mode_Select.1
		THEN
			In_Auto:= FALSE;
			In_Auto_Mode:= FALSE;
	END_IF;
	In_Manual:= NOT In_Auto;
	In_Manual_Mode:= In_Manual;

(*--------------------------------------------------------------------------------Tool Positions---------------------------------------------------------------*)
	Tool_States();

(*----------------------------------------------------Part Present Sensor Input Patterns----------------------------------------------------------------*)
	All_Sensors();


(*>>>>>>>>>>>>>>>>>>>>>>>>>>>>>>>>>>>>>>>>>> Auto Run Cycle >>>>>>>>>>>>>>>>>>>>>>>>>>>>>>>>>>>>>>>*)
(*+++++++++++THIS AREA IS CUSTOM PER INSTALLATION AND WILL HAVE TO BE MODIFIED PER +++++++++++++*)
(*+++++++++++THIS AREA IS CUSTOM PER INSTALLATION AND WILL HAVE TO BE MODIFIED PER +++++++++++++*)
	(*Control of Auto_Run*)
	Auto_Run:= Enable_Motion AND In_Auto AND Model_ID<>0 AND NOT Cycle_Complete;

	(*Auto Run Enables All Other Auto Cycle Code*)
	IF Auto_Run
		THEN

			IF (NOT Load_Complete1 OR (Load_Robots_UnclampEarly1 AND All_Sensors_On.1))
				AND Load_Robots_Clear2 AND Stud_Robots_Clear AND Seal_Robots_Clear
				AND Weld_Robots_Clear AND TurnTable_Clear AND Unload_Robots_Clear
				AND TurnTableA_At_Robot
				THEN
					(*Start 1st Load Robots*)
					Start_Load_Robots1:= ((Tool_At_Load.0 AND All_Sensors_Off AND NOT Repo_Reqs.0 AND Load_Robots_PartInEOAT1)
									OR (Tool_At_Load.1 AND All_Sensors_On.4 AND Repo_Reqs.0))
									OR Load_Robots_WorkingOK1;
					(*Allow 1st Load Robots To Proceed*)
					Load_Robots_Proceed1:= Tool_At_Load.0 AND All_Sensors_Off AND Load_Robots_PartInEOAT1;
			ELSE
					Start_Load_Robots1:= FALSE;
					Load_Robots_Proceed1:= FALSE;
			END_IF;


			IF (NOT Load_Complete2 OR (Load_Robots_UnclampEarly2 AND All_Sensors_On.2))
				AND Load_Robots_Clear1 AND Stud_Robots_Clear AND Seal_Robots_Clear
				AND Weld_Robots_Clear AND TurnTable_Clear AND Unload_Robots_Clear
				AND TurnTableA_At_Robot
				THEN
					(*Start 2nd Load Robots*)
					Start_Load_Robots2:= ((Tool_At_Load.1 AND All_Sensors_Off AND NOT Repo_Reqs.0 AND Load_Robots_PartInEOAT2)
									OR (Tool_At_Load.1 AND All_Sensors_On.4 AND Repo_Reqs.0))
									OR Load_Robots_WorkingOK2;
					(*Allow 2nd Load Robots To Proceed*)
					Load_Robots_Proceed2:= Tool_At_Load.1 AND All_Sensors_Off AND Load_Robots_PartInEOAT2;
			ELSE
					Start_Load_Robots2:= FALSE;
					Load_Robots_Proceed2:= FALSE;
			END_IF;


